  STRUCT
   S700_PLT : STRUCT 	//Temporary placeholder variable
    RACK0_PLT_CODE : INT ;
    RACK0_PLT_QTY : INT ;
    RACK0_PLT_PRIORITY : INT ;
    RACK0_HMI_PLT_CODE : INT ;
    RACK0_HMI_PLT_QTY : INT ;
    RACK1_PLT_CODE : INT ;
    RACK1_PLT_QTY : INT ;
    RACK1_PLT_PRIORITY : INT ;
    RACK1_HMI_PLT_CODE : INT ;
    RACK1_HMI_PLT_QTY : INT ;
    RACK2_PLT_CODE : INT ;
    RACK2_PLT_QTY : INT ;
    RACK2_PLT_PRIORITY : INT ;
    RACK2_HMI_PLT_CODE : INT ;
    RACK2_HMI_PLT_QTY : INT ;
    RACK3_PLT_CODE : INT ;
    RACK3_PLT_QTY : INT ;
    RACK3_PLT_PRIORITY : INT ;
    RACK3_HMI_PLT_CODE : INT ;
    RACK3_HMI_PLT_QTY : INT ;
    RACK4_PLT_CODE : INT ;
    RACK4_PLT_QTY : INT ;
    RACK4_PLT_PRIORITY : INT ;
    RACK4_HMI_PLT_CODE : INT ;
    RACK4_HMI_PLT_QTY : INT ;
    RACK5_PLT_CODE : INT ;
    RACK5_PLT_QTY : INT ;
    RACK5_PLT_PRIORITY : INT ;
    RACK5_HMI_PLT_CODE : INT ;
    RACK5_HMI_PLT_QTY : INT ;
    RACK6_PLT_CODE : INT ;
    RACK6_PLT_QTY : INT ;
    RACK6_PLT_PRIORITY : INT ;
    RACK6_HMI_PLT_CODE : INT ;
    RACK6_HMI_PLT_QTY : INT ;
    RACK7_PLT_CODE : INT ;
    RACK7_PLT_QTY : INT ;
    RACK7_PLT_PRIORITY : INT ;
    RACK7_HMI_PLT_CODE : INT ;
    RACK7_HMI_PLT_QTY : INT ;
    RACK8_PLT_CODE : INT ;
    RACK8_PLT_QTY : INT ;
    RACK8_PLT_PRIORITY : INT ;
    RACK8_HMI_PLT_CODE : INT ;
    RACK8_HMI_PLT_QTY : INT ;
    RACK9_PLT_CODE : INT ;
    RACK9_PLT_QTY : INT ;
    RACK9_PLT_PRIORITY : INT ;
    RACK9_HMI_PLT_CODE : INT ;
    RACK9_HMI_PLT_QTY : INT ;
    RACK10_PLT_CODE : INT ;
    RACK10_PLT_QTY : INT ;
    RACK10_PLT_PRIORITY : INT ;
    RACK10_HMI_PLT_CODE : INT ;
    RACK10_HMI_PLT_QTY : INT ;
    RACK11_PLT_CODE : INT ;
    RACK11_PLT_QTY : INT ;
    RACK11_PLT_PRIORITY : INT ;
    RACK11_HMI_PLT_CODE : INT ;
    RACK11_HMI_PLT_QTY : INT ;
    RACK12_PLT_CODE : INT ;
    RACK12_PLT_QTY : INT ;
    RACK12_PLT_PRIORITY : INT ;
    RACK12_HMI_PLT_CODE : INT ;
    RACK12_HMI_PLT_QTY : INT ;
   END_STRUCT ;
  END_STRUCT ;
BEGIN
   S700_PLT.RACK0_PLT_CODE := 0;
   S700_PLT.RACK0_PLT_QTY := 0;
   S700_PLT.RACK0_PLT_PRIORITY := 0;
   S700_PLT.RACK0_HMI_PLT_CODE := 0;
   S700_PLT.RACK0_HMI_PLT_QTY := 0;
   S700_PLT.RACK1_PLT_CODE := 0;
   S700_PLT.RACK1_PLT_QTY := 0;
   S700_PLT.RACK1_PLT_PRIORITY := 0;
   S700_PLT.RACK1_HMI_PLT_CODE := 0;
   S700_PLT.RACK1_HMI_PLT_QTY := 0;
   S700_PLT.RACK2_PLT_CODE := 0;
   S700_PLT.RACK2_PLT_QTY := 0;
   S700_PLT.RACK2_PLT_PRIORITY := 0;
   S700_PLT.RACK2_HMI_PLT_CODE := 0;
   S700_PLT.RACK2_HMI_PLT_QTY := 0;
   S700_PLT.RACK3_PLT_CODE := 0;
   S700_PLT.RACK3_PLT_QTY := 0;
   S700_PLT.RACK3_PLT_PRIORITY := 0;
   S700_PLT.RACK3_HMI_PLT_CODE := 0;
   S700_PLT.RACK3_HMI_PLT_QTY := 0;
   S700_PLT.RACK4_PLT_CODE := 0;
   S700_PLT.RACK4_PLT_QTY := 0;
   S700_PLT.RACK4_PLT_PRIORITY := 0;
   S700_PLT.RACK4_HMI_PLT_CODE := 0;
   S700_PLT.RACK4_HMI_PLT_QTY := 0;
   S700_PLT.RACK5_PLT_CODE := 0;
   S700_PLT.RACK5_PLT_QTY := 0;
   S700_PLT.RACK5_PLT_PRIORITY := 0;
   S700_PLT.RACK5_HMI_PLT_CODE := 0;
   S700_PLT.RACK5_HMI_PLT_QTY := 0;
   S700_PLT.RACK6_PLT_CODE := 0;
   S700_PLT.RACK6_PLT_QTY := 0;
   S700_PLT.RACK6_PLT_PRIORITY := 0;
   S700_PLT.RACK6_HMI_PLT_CODE := 0;
   S700_PLT.RACK6_HMI_PLT_QTY := 0;
   S700_PLT.RACK7_PLT_CODE := 0;
   S700_PLT.RACK7_PLT_QTY := 0;
   S700_PLT.RACK7_PLT_PRIORITY := 0;
   S700_PLT.RACK7_HMI_PLT_CODE := 0;
   S700_PLT.RACK7_HMI_PLT_QTY := 0;
   S700_PLT.RACK8_PLT_CODE := 0;
   S700_PLT.RACK8_PLT_QTY := 0;
   S700_PLT.RACK8_PLT_PRIORITY := 0;
   S700_PLT.RACK8_HMI_PLT_CODE := 0;
   S700_PLT.RACK8_HMI_PLT_QTY := 0;
   S700_PLT.RACK9_PLT_CODE := 0;
   S700_PLT.RACK9_PLT_QTY := 0;
   S700_PLT.RACK9_PLT_PRIORITY := 0;
   S700_PLT.RACK9_HMI_PLT_CODE := 0;
   S700_PLT.RACK9_HMI_PLT_QTY := 0;
   S700_PLT.RACK10_PLT_CODE := 0;
   S700_PLT.RACK10_PLT_QTY := 0;
   S700_PLT.RACK10_PLT_PRIORITY := 0;
   S700_PLT.RACK10_HMI_PLT_CODE := 0;
   S700_PLT.RACK10_HMI_PLT_QTY := 0;
   S700_PLT.RACK11_PLT_CODE := 0;
   S700_PLT.RACK11_PLT_QTY := 0;
   S700_PLT.RACK11_PLT_PRIORITY := 0;
   S700_PLT.RACK11_HMI_PLT_CODE := 0;
   S700_PLT.RACK11_HMI_PLT_QTY := 0;
   S700_PLT.RACK12_PLT_CODE := 0;
   S700_PLT.RACK12_PLT_QTY := 0;
   S700_PLT.RACK12_PLT_PRIORITY := 0;
   S700_PLT.RACK12_HMI_PLT_CODE := 0;
   S700_PLT.RACK12_HMI_PLT_QTY := 0;
END_DATA_BLOCK

DATA_BLOCK DB 60
TITLE =
VERSION : 0.1


  STRUCT
   FC1_SEND_1 : ARRAY  [0 .. 699 ] OF BYTE  := B#16#0;
  END_STRUCT ;
BEGIN
   FC1_SEND_1[0] := B#16#0;
   FC1_SEND_1[1] := B#16#0;
   FC1_SEND_1[2] := B#16#0;
   FC1_SEND_1[3] := B#16#0;
   FC1_SEND_1[4] := B#16#0;
   FC1_SEND_1[5] := B#16#0;
   FC1_SEND_1[6] := B#16#0;
   FC1_SEND_1[7] := B#16#0;
   FC1_SEND_1[8] := B#16#0;
   FC1_SEND_1[9] := B#16#0;
   FC1_SEND_1[10] := B#16#0;
   FC1_SEND_1[11] := B#16#0;
   FC1_SEND_1[12] := B#16#0;
   FC1_SEND_1[13] := B#16#0;
   FC1_SEND_1[14] := B#16#0;
   FC1_SEND_1[15] := B#16#0;
   FC1_SEND_1[16] := B#16#0;
   FC1_SEND_1[17] := B#16#0;
   FC1_SEND_1[18] := B#16#0;
   FC1_SEND_1[19] := B#16#0;
   FC1_SEND_1[20] := B#16#0;
   FC1_SEND_1[21] := B#16#0;
   FC1_SEND_1[22] := B#16#0;
   FC1_SEND_1[23] := B#16#0;
   FC1_SEND_1[24] := B#16#0;
   FC1_SEND_1[25] := B#16#0;
   FC1_SEND_1[26] := B#16#0;
   FC1_SEND_1[27] := B#16#0;
   FC1_SEND_1[28] := B#16#0;
   FC1_SEND_1[29] := B#16#0;
   FC1_SEND_1[30] := B#16#0;
   FC1_SEND_1[31] := B#16#0;
   FC1_SEND_1[32] := B#16#0;
   FC1_SEND_1[33] := B#16#0;
   FC1_SEND_1[34] := B#16#0;
   FC1_SEND_1[35] := B#16#0;
   FC1_SEND_1[36] := B#16#0;
   FC1_SEND_1[37] := B#16#0;
   FC1_SEND_1[38] := B#16#0;
   FC1_SEND_1[39] := B#16#0;
   FC1_SEND_1[40] := B#16#0;
   FC1_SEND_1[41] := B#16#0;
   FC1_SEND_1[42] := B#16#0;
   FC1_SEND_1[43] := B#16#0;
   FC1_SEND_1[44] := B#16#0;
   FC1_SEND_1[45] := B#16#0;
   FC1_SEND_1[46] := B#16#0;
   FC1_SEND_1[47] := B#16#0;
   FC1_SEND_1[48] := B#16#0;
   FC1_SEND_1[49] := B#16#0;
   FC1_SEND_1[50] := B#16#0;
   FC1_SEND_1[51] := B#16#0;
   FC1_SEND_1[52] := B#16#0;
   FC1_SEND_1[53] := B#16#0;
   FC1_SEND_1[54] := B#16#0;
   FC1_SEND_1[55] := B#16#0;
   FC1_SEND_1[56] := B#16#0;
   FC1_SEND_1[57] := B#16#0;
   FC1_SEND_1[58] := B#16#0;
   FC1_SEND_1[59] := B#16#0;
   FC1_SEND_1[60] := B#16#0;
   FC1_SEND_1[61] := B#16#0;
   FC1_SEND_1[62] := B#16#0;
   FC1_SEND_1[63] := B#16#0;
   FC1_SEND_1[64] := B#16#0;
   FC1_SEND_1[65] := B#16#0;
   FC1_SEND_1[66] := B#16#0;
   FC1_SEND_1[67] := B#16#0;
   FC1_SEND_1[68] := B#16#0;
   FC1_SEND_1[69] := B#16#0;
   FC1_SEND_1[70] := B#16#0;
   FC1_SEND_1[71] := B#16#0;
   FC1_SEND_1[72] := B#16#0;
   FC1_SEND_1[73] := B#16#0;
   FC1_SEND_1[74] := B#16#0;
   FC1_SEND_1[75] := B#16#0;
   FC1_SEND_1[76] := B#16#0;
   FC1_SEND_1[77] := B#16#0;
   FC1_SEND_1[78] := B#16#0;
   FC1_SEND_1[79] := B#16#0;
   FC1_SEND_1[80] := B#16#0;
   FC1_SEND_1[81] := B#16#0;
   FC1_SEND_1[82] := B#16#0;
   FC1_SEND_1[83] := B#16#0;
   FC1_SEND_1[84] := B#16#0;
   FC1_SEND_1[85] := B#16#0;
   FC1_SEND_1[86] := B#16#0;
   FC1_SEND_1[87] := B#16#0;
   FC1_SEND_1[88] := B#16#0;
   FC1_SEND_1[89] := B#16#0;
   FC1_SEND_1[90] := B#16#0;
   FC1_SEND_1[91] := B#16#0;
   FC1_SEND_1[92] := B#16#0;
   FC1_SEND_1[93] := B#16#0;
   FC1_SEND_1[94] := B#16#0;
   FC1_SEND_1[95] := B#16#0;
   FC1_SEND_1[96] := B#16#0;
   FC1_SEND_1[97] := B#16#0;
   FC1_SEND_1[98] := B#16#0;
   FC1_SEND_1[99] := B#16#0;
   FC1_SEND_1[100] := B#16#0;
   FC1_SEND_1[101] := B#16#0;
   FC1_SEND_1[102] := B#16#0;
   FC1_SEND_1[103] := B#16#0;
   FC1_SEND_1[104] := B#16#0;
   FC1_SEND_1[105] := B#16#0;
   FC1_SEND_1[106] := B#16#0;
   FC1_SEND_1[107] := B#16#0;
   FC1_SEND_1[108] := B#16#0;
   FC1_SEND_1[109] := B#16#0;
   FC1_SEND_1[110] := B#16#0;
   FC1_SEND_1[111] := B#16#0;
   FC1_SEND_1[112] := B#16#0;
   FC1_SEND_1[113] := B#16#0;
   FC1_SEND_1[114] := B#16#0;
   FC1_SEND_1[115] := B#16#0;
   FC1_SEND_1[116] := B#16#0;
   FC1_SEND_1[117] := B#16#0;
   FC1_SEND_1[118] := B#16#0;
   FC1_SEND_1[119] := B#16#0;
   FC1_SEND_1[120] := B#16#0;
   FC1_SEND_1[121] := B#16#0;
   FC1_SEND_1[122] := B#16#0;
   FC1_SEND_1[123] := B#16#0;
   FC1_SEND_1[124] := B#16#0;
   FC1_SEND_1[125] := B#16#0;
   FC1_SEND_1[126] := B#16#0;
   FC1_SEND_1[127] := B#16#0;
   FC1_SEND_1[128] := B#16#0;
   FC1_SEND_1[129] := B#16#0;
   FC1_SEND_1[130] := B#16#0;
   FC1_SEND_1[131] := B#16#0;
   FC1_SEND_1[132] := B#16#0;
   FC1_SEND_1[133] := B#16#0;
   FC1_SEND_1[134] := B#16#0;
   FC1_SEND_1[135] := B#16#0;
   FC1_SEND_1[136] := B#16#0;
   FC1_SEND_1[137] := B#16#0;
   FC1_SEND_1[138] := B#16#0;
   FC1_SEND_1[139] := B#16#0;
   FC1_SEND_1[140] := B#16#0;
   FC1_SEND_1[141] := B#16#0;
   FC1_SEND_1[142] := B#16#0;
   FC1_SEND_1[143] := B#16#0;
   FC1_SEND_1[144] := B#16#0;
   FC1_SEND_1[145] := B#16#0;
   FC1_SEND_1[146] := B#16#0;
   FC1_SEND_1[147] := B#16#0;
   FC1_SEND_1[148] := B#16#0;
   FC1_SEND_1[149] := B#16#0;
   FC1_SEND_1[150] := B#16#0;
   FC1_SEND_1[151] := B#16#0;
   FC1_SEND_1[152] := B#16#0;
   FC1_SEND_1[153] := B#16#0;
   FC1_SEND_1[154] := B#16#0;
   FC1_SEND_1[155] := B#16#0;
   FC1_SEND_1[156] := B#16#0;
   FC1_SEND_1[157] := B#16#0;
   FC1_SEND_1[158] := B#16#0;
   FC1_SEND_1[159] := B#16#0;
   FC1_SEND_1[160] := B#16#0;
   FC1_SEND_1[161] := B#16#0;
   FC1_SEND_1[162] := B#16#0;
   FC1_SEND_1[163] := B#16#0;
   FC1_SEND_1[164] := B#16#0;
   FC1_SEND_1[165] := B#16#0;
   FC1_SEND_1[166] := B#16#0;
   FC1_SEND_1[167] := B#16#0;
   FC1_SEND_1[168] := B#16#0;
   FC1_SEND_1[169] := B#16#0;
   FC1_SEND_1[170] := B#16#0;
   FC1_SEND_1[171] := B#16#0;
   FC1_SEND_1[172] := B#16#0;
   FC1_SEND_1[173] := B#16#0;
   FC1_SEND_1[174] := B#16#0;
   FC1_SEND_1[175] := B#16#0;
   FC1_SEND_1[176] := B#16#0;
   FC1_SEND_1[177] := B#16#0;
   FC1_SEND_1[178] := B#16#0;
   FC1_SEND_1[179] := B#16#0;
   FC1_SEND_1[180] := B#16#0;
   FC1_SEND_1[181] := B#16#0;
   FC1_SEND_1[182] := B#16#0;
   FC1_SEND_1[183] := B#16#0;
   FC1_SEND_1[184] := B#16#0;
   FC1_SEND_1[185] := B#16#0;
   FC1_SEND_1[186] := B#16#0;
   FC1_SEND_1[187] := B#16#0;
   FC1_SEND_1[188] := B#16#0;
   FC1_SEND_1[189] := B#16#0;
   FC1_SEND_1[190] := B#16#0;
   FC1_SEND_1[191] := B#16#0;
   FC1_SEND_1[192] := B#16#0;
   FC1_SEND_1[193] := B#16#0;
   FC1_SEND_1[194] := B#16#0;
   FC1_SEND_1[195] := B#16#0;
   FC1_SEND_1[196] := B#16#0;
   FC1_SEND_1[197] := B#16#0;
   FC1_SEND_1[198] := B#16#0;
   FC1_SEND_1[199] := B#16#0;
   FC1_SEND_1[200] := B#16#0;
   FC1_SEND_1[201] := B#16#0;
   FC1_SEND_1[202] := B#16#0;
   FC1_SEND_1[203] := B#16#0;
   FC1_SEND_1[204] := B#16#0;
   FC1_SEND_1[205] := B#16#0;
   FC1_SEND_1[206] := B#16#0;
   FC1_SEND_1[207] := B#16#0;
   FC1_SEND_1[208] := B#16#0;
   FC1_SEND_1[209] := B#16#0;
   FC1_SEND_1[210] := B#16#0;
   FC1_SEND_1[211] := B#16#0;
   FC1_SEND_1[212] := B#16#0;
   FC1_SEND_1[213] := B#16#0;
   FC1_SEND_1[214] := B#16#0;
   FC1_SEND_1[215] := B#16#0;
   FC1_SEND_1[216] := B#16#0;
   FC1_SEND_1[217] := B#16#0;
   FC1_SEND_1[218] := B#16#0;
   FC1_SEND_1[219] := B#16#0;
   FC1_SEND_1[220] := B#16#0;
   FC1_SEND_1[221] := B#16#0;
   FC1_SEND_1[222] := B#16#0;
   FC1_SEND_1[223] := B#16#0;
   FC1_SEND_1[224] := B#16#0;
   FC1_SEND_1[225] := B#16#0;
   FC1_SEND_1[226] := B#16#0;
   FC1_SEND_1[227] := B#16#0;
   FC1_SEND_1[228] := B#16#0;
   FC1_SEND_1[229] := B#16#0;
   FC1_SEND_1[230] := B#16#0;
   FC1_SEND_1[231] := B#16#0;
   FC1_SEND_1[232] := B#16#0;
   FC1_SEND_1[233] := B#16#0;
   FC1_SEND_1[234] := B#16#0;
   FC1_SEND_1[235] := B#16#0;
   FC1_SEND_1[236] := B#16#0;
   FC1_SEND_1[237] := B#16#0;
   FC1_SEND_1[238] := B#16#0;
   FC1_SEND_1[239] := B#16#0;
   FC1_SEND_1[240] := B#16#0;
   FC1_SEND_1[241] := B#16#0;
   FC1_SEND_1[242] := B#16#0;
   FC1_SEND_1[243] := B#16#0;
   FC1_SEND_1[244] := B#16#0;
   FC1_SEND_1[245] := B#16#0;
   FC1_SEND_1[246] := B#16#0;
   FC1_SEND_1[247] := B#16#0;
   FC1_SEND_1[248] := B#16#0;
   FC1_SEND_1[249] := B#16#0;
   FC1_SEND_1[250] := B#16#0;
   FC1_SEND_1[251] := B#16#0;
   FC1_SEND_1[252] := B#16#0;
   FC1_SEND_1[253] := B#16#0;
   FC1_SEND_1[254] := B#16#0;
   FC1_SEND_1[255] := B#16#0;
   FC1_SEND_1[256] := B#16#0;
   FC1_SEND_1[257] := B#16#0;
   FC1_SEND_1[258] := B#16#0;
   FC1_SEND_1[259] := B#16#0;
   FC1_SEND_1[260] := B#16#0;
   FC1_SEND_1[261] := B#16#0;
   FC1_SEND_1[262] := B#16#0;
   FC1_SEND_1[263] := B#16#0;
   FC1_SEND_1[264] := B#16#0;
   FC1_SEND_1[265] := B#16#0;
   FC1_SEND_1[266] := B#16#0;
   FC1_SEND_1[267] := B#16#0;
   FC1_SEND_1[268] := B#16#0;
   FC1_SEND_1[269] := B#16#0;
   FC1_SEND_1[270] := B#16#0;
   FC1_SEND_1[271] := B#16#0;
   FC1_SEND_1[272] := B#16#0;
   FC1_SEND_1[273] := B#16#0;
   FC1_SEND_1[274] := B#16#0;
   FC1_SEND_1[275] := B#16#0;
   FC1_SEND_1[276] := B#16#0;
   FC1_SEND_1[277] := B#16#0;
   FC1_SEND_1[278] := B#16#0;
   FC1_SEND_1[279] := B#16#0;
   FC1_SEND_1[280] := B#16#0;
   FC1_SEND_1[281] := B#16#0;
   FC1_SEND_1[282] := B#16#0;
   FC1_SEND_1[283] := B#16#0;
   FC1_SEND_1[284] := B#16#0;
   FC1_SEND_1[285] := B#16#0;
   FC1_SEND_1[286] := B#16#0;
   FC1_SEND_1[287] := B#16#0;
   FC1_SEND_1[288] := B#16#0;
   FC1_SEND_1[289] := B#16#0;
   FC1_SEND_1[290] := B#16#0;
   FC1_SEND_1[291] := B#16#0;
   FC1_SEND_1[292] := B#16#0;
   FC1_SEND_1[293] := B#16#0;
   FC1_SEND_1[294] := B#16#0;
   FC1_SEND_1[295] := B#16#0;
   FC1_SEND_1[296] := B#16#0;
   FC1_SEND_1[297] := B#16#0;
   FC1_SEND_1[298] := B#16#0;
   FC1_SEND_1[299] := B#16#0;
   FC1_SEND_1[300] := B#16#0;
   FC1_SEND_1[301] := B#16#0;
   FC1_SEND_1[302] := B#16#0;
   FC1_SEND_1[303] := B#16#0;
   FC1_SEND_1[304] := B#16#0;
   FC1_SEND_1[305] := B#16#0;
   FC1_SEND_1[306] := B#16#0;
   FC1_SEND_1[307] := B#16#0;
   FC1_SEND_1[308] := B#16#0;
   FC1_SEND_1[309] := B#16#0;
   FC1_SEND_1[310] := B#16#0;
   FC1_SEND_1[311] := B#16#0;
   FC1_SEND_1[312] := B#16#0;
   FC1_SEND_1[313] := B#16#0;
   FC1_SEND_1[314] := B#16#0;
   FC1_SEND_1[315] := B#16#0;
   FC1_SEND_1[316] := B#16#0;
   FC1_SEND_1[317] := B#16#0;
   FC1_SEND_1[318] := B#16#0;
   FC1_SEND_1[319] := B#16#0;
   FC1_SEND_1[320] := B#16#0;
   FC1_SEND_1[321] := B#16#0;
   FC1_SEND_1[322] := B#16#0;
   FC1_SEND_1[323] := B#16#0;
   FC1_SEND_1[324] := B#16#0;
   FC1_SEND_1[325] := B#16#0;
   FC1_SEND_1[326] := B#16#0;
   FC1_SEND_1[327] := B#16#0;
   FC1_SEND_1[328] := B#16#0;
   FC1_SEND_1[329] := B#16#0;
   FC1_SEND_1[330] := B#16#0;
   FC1_SEND_1[331] := B#16#0;
   FC1_SEND_1[332] := B#16#0;
   FC1_SEND_1[333] := B#16#0;
   FC1_SEND_1[334] := B#16#0;
   FC1_SEND_1[335] := B#16#0;
   FC1_SEND_1[336] := B#16#0;
   FC1_SEND_1[337] := B#16#0;
   FC1_SEND_1[338] := B#16#0;
   FC1_SEND_1[339] := B#16#0;
   FC1_SEND_1[340] := B#16#0;
   FC1_SEND_1[341] := B#16#0;
   FC1_SEND_1[342] := B#16#0;
   FC1_SEND_1[343] := B#16#0;
   FC1_SEND_1[344] := B#16#0;
   FC1_SEND_1[345] := B#16#0;
   FC1_SEND_1[346] := B#16#0;
   FC1_SEND_1[347] := B#16#0;
   FC1_SEND_1[348] := B#16#0;
   FC1_SEND_1[349] := B#16#0;
   FC1_SEND_1[350] := B#16#0;
   FC1_SEND_1[351] := B#16#0;
   FC1_SEND_1[352] := B#16#0;
   FC1_SEND_1[353] := B#16#0;
   FC1_SEND_1[354] := B#16#0;
   FC1_SEND_1[355] := B#16#0;
   FC1_SEND_1[356] := B#16#0;
   FC1_SEND_1[357] := B#16#0;
   FC1_SEND_1[358] := B#16#0;
   FC1_SEND_1[359] := B#16#0;
   FC1_SEND_1[360] := B#16#0;
   FC1_SEND_1[361] := B#16#0;
   FC1_SEND_1[362] := B#16#0;
   FC1_SEND_1[363] := B#16#0;
   FC1_SEND_1[364] := B#16#0;
   FC1_SEND_1[365] := B#16#0;
   FC1_SEND_1[366] := B#16#0;
   FC1_SEND_1[367] := B#16#0;
   FC1_SEND_1[368] := B#16#0;
   FC1_SEND_1[369] := B#16#0;
   FC1_SEND_1[370] := B#16#0;
   FC1_SEND_1[371] := B#16#0;
   FC1_SEND_1[372] := B#16#0;
   FC1_SEND_1[373] := B#16#0;
   FC1_SEND_1[374] := B#16#0;
   FC1_SEND_1[375] := B#16#0;
   FC1_SEND_1[376] := B#16#0;
   FC1_SEND_1[377] := B#16#0;
   FC1_SEND_1[378] := B#16#0;
   FC1_SEND_1[379] := B#16#0;
   FC1_SEND_1[380] := B#16#0;
   FC1_SEND_1[381] := B#16#0;
   FC1_SEND_1[382] := B#16#0;
   FC1_SEND_1[383] := B#16#0;
   FC1_SEND_1[384] := B#16#0;
   FC1_SEND_1[385] := B#16#0;
   FC1_SEND_1[386] := B#16#0;
   FC1_SEND_1[387] := B#16#0;
   FC1_SEND_1[388] := B#16#0;
   FC1_SEND_1[389] := B#16#0;
   FC1_SEND_1[390] := B#16#0;
   FC1_SEND_1[391] := B#16#0;
   FC1_SEND_1[392] := B#16#0;
   FC1_SEND_1[393] := B#16#0;
   FC1_SEND_1[394] := B#16#0;
   FC1_SEND_1[395] := B#16#0;
   FC1_SEND_1[396] := B#16#0;
   FC1_SEND_1[397] := B#16#0;
   FC1_SEND_1[398] := B#16#0;
   FC1_SEND_1[399] := B#16#0;
   FC1_SEND_1[400] := B#16#0;
   FC1_SEND_1[401] := B#16#0;
   FC1_SEND_1[402] := B#16#0;
   FC1_SEND_1[403] := B#16#0;
   FC1_SEND_1[404] := B#16#0;
   FC1_SEND_1[405] := B#16#0;
   FC1_SEND_1[406] := B#16#0;
   FC1_SEND_1[407] := B#16#0;
   FC1_SEND_1[408] := B#16#0;
   FC1_SEND_1[409] := B#16#0;
   FC1_SEND_1[410] := B#16#0;
   FC1_SEND_1[411] := B#16#0;
   FC1_SEND_1[412] := B#16#0;
   FC1_SEND_1[413] := B#16#0;
   FC1_SEND_1[414] := B#16#0;
   FC1_SEND_1[415] := B#16#0;
   FC1_SEND_1[416] := B#16#0;
   FC1_SEND_1[417] := B#16#0;
   FC1_SEND_1[418] := B#16#0;
   FC1_SEND_1[419] := B#16#0;
   FC1_SEND_1[420] := B#16#0;
   FC1_SEND_1[421] := B#16#0;
   FC1_SEND_1[422] := B#16#0;
   FC1_SEND_1[423] := B#16#0;
   FC1_SEND_1[424] := B#16#0;
   FC1_SEND_1[425] := B#16#0;
   FC1_SEND_1[426] := B#16#0;
   FC1_SEND_1[427] := B#16#0;
   FC1_SEND_1[428] := B#16#0;
   FC1_SEND_1[429] := B#16#0;
   FC1_SEND_1[430] := B#16#0;
   FC1_SEND_1[431] := B#16#0;
   FC1_SEND_1[432] := B#16#0;
   FC1_SEND_1[433] := B#16#0;
   FC1_SEND_1[434] := B#16#0;
   FC1_SEND_1[435] := B#16#0;
   FC1_SEND_1[436] := B#16#0;
   FC1_SEND_1[437] := B#16#0;
   FC1_SEND_1[438] := B#16#0;
   FC1_SEND_1[439] := B#16#0;
   FC1_SEND_1[440] := B#16#0;
   FC1_SEND_1[441] := B#16#0;
   FC1_SEND_1[442] := B#16#0;
   FC1_SEND_1[443] := B#16#0;
   FC1_SEND_1[444] := B#16#0;
   FC1_SEND_1[445] := B#16#0;
   FC1_SEND_1[446] := B#16#0;
   FC1_SEND_1[447] := B#16#0;
   FC1_SEND_1[448] := B#16#0;
   FC1_SEND_1[449] := B#16#0;
   FC1_SEND_1[450] := B#16#0;
   FC1_SEND_1[451] := B#16#0;
   FC1_SEND_1[452] := B#16#0;
   FC1_SEND_1[453] := B#16#0;
   FC1_SEND_1[454] := B#16#0;
   FC1_SEND_1[455] := B#16#0;
   FC1_SEND_1[456] := B#16#0;
   FC1_SEND_1[457] := B#16#0;
   FC1_SEND_1[458] := B#16#0;
   FC1_SEND_1[459] := B#16#0;
   FC1_SEND_1[460] := B#16#0;
   FC1_SEND_1[461] := B#16#0;
   FC1_SEND_1[462] := B#16#0;
   FC1_SEND_1[463] := B#16#0;
   FC1_SEND_1[464] := B#16#0;
   FC1_SEND_1[465] := B#16#0;
   FC1_SEND_1[466] := B#16#0;
   FC1_SEND_1[467] := B#16#0;
   FC1_SEND_1[468] := B#16#0;
   FC1_SEND_1[469] := B#16#0;
   FC1_SEND_1[470] := B#16#0;
   FC1_SEND_1[471] := B#16#0;
   FC1_SEND_1[472] := B#16#0;
   FC1_SEND_1[473] := B#16#0;
   FC1_SEND_1[474] := B#16#0;
   FC1_SEND_1[475] := B#16#0;
   FC1_SEND_1[476] := B#16#0;
   FC1_SEND_1[477] := B#16#0;
   FC1_SEND_1[478] := B#16#0;
   FC1_SEND_1[479] := B#16#0;
   FC1_SEND_1[480] := B#16#0;
   FC1_SEND_1[481] := B#16#0;
   FC1_SEND_1[482] := B#16#0;
   FC1_SEND_1[483] := B#16#0;
   FC1_SEND_1[484] := B#16#0;
   FC1_SEND_1[485] := B#16#0;
   FC1_SEND_1[486] := B#16#0;
   FC1_SEND_1[487] := B#16#0;
   FC1_SEND_1[488] := B#16#0;
   FC1_SEND_1[489] := B#16#0;
   FC1_SEND_1[490] := B#16#0;
   FC1_SEND_1[491] := B#16#0;
   FC1_SEND_1[492] := B#16#0;
   FC1_SEND_1[493] := B#16#0;
   FC1_SEND_1[494] := B#16#0;
   FC1_SEND_1[495] := B#16#0;
   FC1_SEND_1[496] := B#16#0;
   FC1_SEND_1[497] := B#16#0;
   FC1_SEND_1[498] := B#16#0;
   FC1_SEND_1[499] := B#16#0;
   FC1_SEND_1[500] := B#16#0;
   FC1_SEND_1[501] := B#16#0;
   FC1_SEND_1[502] := B#16#0;
   FC1_SEND_1[503] := B#16#0;
   FC1_SEND_1[504] := B#16#0;
   FC1_SEND_1[505] := B#16#0;
   FC1_SEND_1[506] := B#16#0;
   FC1_SEND_1[507] := B#16#0;
   FC1_SEND_1[508] := B#16#0;
   FC1_SEND_1[509] := B#16#0;
   FC1_SEND_1[510] := B#16#0;
   FC1_SEND_1[511] := B#16#0;
   FC1_SEND_1[512] := B#16#0;
   FC1_SEND_1[513] := B#16#0;
   FC1_SEND_1[514] := B#16#0;
   FC1_SEND_1[515] := B#16#0;
   FC1_SEND_1[516] := B#16#0;
   FC1_SEND_1[517] := B#16#0;
   FC1_SEND_1[518] := B#16#0;
   FC1_SEND_1[519] := B#16#0;
   FC1_SEND_1[520] := B#16#0;
   FC1_SEND_1[521] := B#16#0;
   FC1_SEND_1[522] := B#16#0;
   FC1_SEND_1[523] := B#16#0;
   FC1_SEND_1[524] := B#16#0;
   FC1_SEND_1[525] := B#16#0;
   FC1_SEND_1[526] := B#16#0;
   FC1_SEND_1[527] := B#16#0;
   FC1_SEND_1[528] := B#16#0;
   FC1_SEND_1[529] := B#16#0;
   FC1_SEND_1[530] := B#16#0;
   FC1_SEND_1[531] := B#16#0;
   FC1_SEND_1[532] := B#16#0;
   FC1_SEND_1[533] := B#16#0;
   FC1_SEND_1[534] := B#16#0;
   FC1_SEND_1[535] := B#16#0;
   FC1_SEND_1[536] := B#16#0;
   FC1_SEND_1[537] := B#16#0;
   FC1_SEND_1[538] := B#16#0;
   FC1_SEND_1[539] := B#16#0;
   FC1_SEND_1[540] := B#16#0;
   FC1_SEND_1[541] := B#16#0;
   FC1_SEND_1[542] := B#16#0;
   FC1_SEND_1[543] := B#16#0;
   FC1_SEND_1[544] := B#16#0;
   FC1_SEND_1[545] := B#16#0;
   FC1_SEND_1[546] := B#16#0;
   FC1_SEND_1[547] := B#16#0;
   FC1_SEND_1[548] := B#16#0;
   FC1_SEND_1[549] := B#16#0;
   FC1_SEND_1[550] := B#16#0;
   FC1_SEND_1[551] := B#16#0;
   FC1_SEND_1[552] := B#16#0;
   FC1_SEND_1[553] := B#16#0;
   FC1_SEND_1[554] := B#16#0;
   FC1_SEND_1[555] := B#16#0;
   FC1_SEND_1[556] := B#16#0;
   FC1_SEND_1[557] := B#16#0;
   FC1_SEND_1[558] := B#16#0;
   FC1_SEND_1[559] := B#16#0;
   FC1_SEND_1[560] := B#16#0;
   FC1_SEND_1[561] := B#16#0;
   FC1_SEND_1[562] := B#16#0;
   FC1_SEND_1[563] := B#16#0;
   FC1_SEND_1[564] := B#16#0;
   FC1_SEND_1[565] := B#16#0;
   FC1_SEND_1[566] := B#16#0;
   FC1_SEND_1[567] := B#16#0;
   FC1_SEND_1[568] := B#16#0;
   FC1_SEND_1[569] := B#16#0;
   FC1_SEND_1[570] := B#16#0;
   FC1_SEND_1[571] := B#16#0;
   FC1_SEND_1[572] := B#16#0;
   FC1_SEND_1[573] := B#16#0;
   FC1_SEND_1[574] := B#16#0;
   FC1_SEND_1[575] := B#16#0;
   FC1_SEND_1[576] := B#16#0;
   FC1_SEND_1[577] := B#16#0;
   FC1_SEND_1[578] := B#16#0;
   FC1_SEND_1[579] := B#16#0;
   FC1_SEND_1[580] := B#16#0;
   FC1_SEND_1[581] := B#16#0;
   FC1_SEND_1[582] := B#16#0;
   FC1_SEND_1[583] := B#16#0;
   FC1_SEND_1[584] := B#16#0;
   FC1_SEND_1[585] := B#16#0;
   FC1_SEND_1[586] := B#16#0;
   FC1_SEND_1[587] := B#16#0;
   FC1_SEND_1[588] := B#16#0;
   FC1_SEND_1[589] := B#16#0;
   FC1_SEND_1[590] := B#16#0;
   FC1_SEND_1[591] := B#16#0;
   FC1_SEND_1[592] := B#16#0;
   FC1_SEND_1[593] := B#16#0;
   FC1_SEND_1[594] := B#16#0;
   FC1_SEND_1[595] := B#16#0;
   FC1_SEND_1[596] := B#16#0;
   FC1_SEND_1[597] := B#16#0;
   FC1_SEND_1[598] := B#16#0;
   FC1_SEND_1[599] := B#16#0;
   FC1_SEND_1[600] := B#16#0;
   FC1_SEND_1[601] := B#16#0;
   FC1_SEND_1[602] := B#16#0;
   FC1_SEND_1[603] := B#16#0;
   FC1_SEND_1[604] := B#16#0;
   FC1_SEND_1[605] := B#16#0;
   FC1_SEND_1[606] := B#16#0;
   FC1_SEND_1[607] := B#16#0;
   FC1_SEND_1[608] := B#16#0;
   FC1_SEND_1[609] := B#16#0;
   FC1_SEND_1[610] := B#16#0;
   FC1_SEND_1[611] := B#16#0;
   FC1_SEND_1[612] := B#16#0;
   FC1_SEND_1[613] := B#16#0;
   FC1_SEND_1[614] := B#16#0;
   FC1_SEND_1[615] := B#16#0;
   FC1_SEND_1[616] := B#16#0;
   FC1_SEND_1[617] := B#16#0;
   FC1_SEND_1[618] := B#16#0;
   FC1_SEND_1[619] := B#16#0;
   FC1_SEND_1[620] := B#16#0;
   FC1_SEND_1[621] := B#16#0;
   FC1_SEND_1[622] := B#16#0;
   FC1_SEND_1[623] := B#16#0;
   FC1_SEND_1[624] := B#16#0;
   FC1_SEND_1[625] := B#16#0;
   FC1_SEND_1[626] := B#16#0;
   FC1_SEND_1[627] := B#16#0;
   FC1_SEND_1[628] := B#16#0;
   FC1_SEND_1[629] := B#16#0;
   FC1_SEND_1[630] := B#16#0;
   FC1_SEND_1[631] := B#16#0;
   FC1_SEND_1[632] := B#16#0;
   FC1_SEND_1[633] := B#16#0;
   FC1_SEND_1[634] := B#16#0;
   FC1_SEND_1[635] := B#16#0;
   FC1_SEND_1[636] := B#16#0;
   FC1_SEND_1[637] := B#16#0;
   FC1_SEND_1[638] := B#16#0;
   FC1_SEND_1[639] := B#16#0;
   FC1_SEND_1[640] := B#16#0;
   FC1_SEND_1[641] := B#16#0;
   FC1_SEND_1[642] := B#16#0;
   FC1_SEND_1[643] := B#16#0;
   FC1_SEND_1[644] := B#16#0;
   FC1_SEND_1[645] := B#16#0;
   FC1_SEND_1[646] := B#16#0;
   FC1_SEND_1[647] := B#16#0;
   FC1_SEND_1[648] := B#16#0;
   FC1_SEND_1[649] := B#16#0;
   FC1_SEND_1[650] := B#16#0;
   FC1_SEND_1[651] := B#16#0;
   FC1_SEND_1[652] := B#16#0;
   FC1_SEND_1[653] := B#16#0;
   FC1_SEND_1[654] := B#16#0;
   FC1_SEND_1[655] := B#16#0;
   FC1_SEND_1[656] := B#16#0;
   FC1_SEND_1[657] := B#16#0;
   FC1_SEND_1[658] := B#16#0;
   FC1_SEND_1[659] := B#16#0;
   FC1_SEND_1[660] := B#16#0;
   FC1_SEND_1[661] := B#16#0;
   FC1_SEND_1[662] := B#16#0;
   FC1_SEND_1[663] := B#16#0;
   FC1_SEND_1[664] := B#16#0;
   FC1_SEND_1[665] := B#16#0;
   FC1_SEND_1[666] := B#16#0;
   FC1_SEND_1[667] := B#16#0;
   FC1_SEND_1[668] := B#16#0;
   FC1_SEND_1[669] := B#16#0;
   FC1_SEND_1[670] := B#16#0;
   FC1_SEND_1[671] := B#16#0;
   FC1_SEND_1[672] := B#16#0;
   FC1_SEND_1[673] := B#16#0;
   FC1_SEND_1[674] := B#16#0;
   FC1_SEND_1[675] := B#16#0;
   FC1_SEND_1[676] := B#16#0;
   FC1_SEND_1[677] := B#16#0;
   FC1_SEND_1[678] := B#16#0;
   FC1_SEND_1[679] := B#16#0;
   FC1_SEND_1[680] := B#16#0;
   FC1_SEND_1[681] := B#16#0;
   FC1_SEND_1[682] := B#16#0;
   FC1_SEND_1[683] := B#16#0;
   FC1_SEND_1[684] := B#16#0;
   FC1_SEND_1[685] := B#16#0;
   FC1_SEND_1[686] := B#16#0;
   FC1_SEND_1[687] := B#16#0;
   FC1_SEND_1[688] := B#16#0;
   FC1_SEND_1[689] := B#16#0;
   FC1_SEND_1[690] := B#16#0;
   FC1_SEND_1[691] := B#16#0;
   FC1_SEND_1[692] := B#16#0;
   FC1_SEND_1[693] := B#16#0;
   FC1_SEND_1[694] := B#16#0;
   FC1_SEND_1[695] := B#16#0;
   FC1_SEND_1[696] := B#16#0;
   FC1_SEND_1[697] := B#16#0;
   FC1_SEND_1[698] := B#16#0;
   FC1_SEND_1[699] := B#16#0;
END_DATA_BLOCK

DATA_BLOCK DB 61
TITLE =
VERSION : 0.1


  STRUCT
   FC2_RECV_1 : ARRAY  [0 .. 699 ] OF BYTE  := B#16#0;
  END_STRUCT ;
BEGIN
   FC2_RECV_1[0] := B#16#0;
   FC2_RECV_1[1] := B#16#0;
   FC2_RECV_1[2] := B#16#0;
   FC2_RECV_1[3] := B#16#0;
   FC2_RECV_1[4] := B#16#0;
   FC2_RECV_1[5] := B#16#0;
   FC2_RECV_1[6] := B#16#0;
   FC2_RECV_1[7] := B#16#0;
   FC2_RECV_1[8] := B#16#0;
   FC2_RECV_1[9] := B#16#0;
   FC2_RECV_1[10] := B#16#0;
   FC2_RECV_1[11] := B#16#0;
   FC2_RECV_1[12] := B#16#0;
   FC2_RECV_1[13] := B#16#0;
   FC2_RECV_1[14] := B#16#0;
   FC2_RECV_1[15] := B#16#0;
   FC2_RECV_1[16] := B#16#0;
   FC2_RECV_1[17] := B#16#0;
   FC2_RECV_1[18] := B#16#0;
   FC2_RECV_1[19] := B#16#0;
   FC2_RECV_1[20] := B#16#0;
   FC2_RECV_1[21] := B#16#0;
   FC2_RECV_1[22] := B#16#0;
   FC2_RECV_1[23] := B#16#0;
   FC2_RECV_1[24] := B#16#0;
   FC2_RECV_1[25] := B#16#0;
   FC2_RECV_1[26] := B#16#0;
   FC2_RECV_1[27] := B#16#0;
   FC2_RECV_1[28] := B#16#0;
   FC2_RECV_1[29] := B#16#0;
   FC2_RECV_1[30] := B#16#0;
   FC2_RECV_1[31] := B#16#0;
   FC2_RECV_1[32] := B#16#0;
   FC2_RECV_1[33] := B#16#0;
   FC2_RECV_1[34] := B#16#0;
   FC2_RECV_1[35] := B#16#0;
   FC2_RECV_1[36] := B#16#0;
   FC2_RECV_1[37] := B#16#0;
   FC2_RECV_1[38] := B#16#0;
   FC2_RECV_1[39] := B#16#0;
   FC2_RECV_1[40] := B#16#0;
   FC2_RECV_1[41] := B#16#0;
   FC2_RECV_1[42] := B#16#0;
   FC2_RECV_1[43] := B#16#0;
   FC2_RECV_1[44] := B#16#0;
   FC2_RECV_1[45] := B#16#0;
   FC2_RECV_1[46] := B#16#0;
   FC2_RECV_1[47] := B#16#0;
   FC2_RECV_1[48] := B#16#0;
   FC2_RECV_1[49] := B#16#0;
   FC2_RECV_1[50] := B#16#0;
   FC2_RECV_1[51] := B#16#0;
   FC2_RECV_1[52] := B#16#0;
   FC2_RECV_1[53] := B#16#0;
   FC2_RECV_1[54] := B#16#0;
   FC2_RECV_1[55] := B#16#0;
   FC2_RECV_1[56] := B#16#0;
   FC2_RECV_1[57] := B#16#0;
   FC2_RECV_1[58] := B#16#0;
   FC2_RECV_1[59] := B#16#0;
   FC2_RECV_1[60] := B#16#0;
   FC2_RECV_1[61] := B#16#0;
   FC2_RECV_1[62] := B#16#0;
   FC2_RECV_1[63] := B#16#0;
   FC2_RECV_1[64] := B#16#0;
   FC2_RECV_1[65] := B#16#0;
   FC2_RECV_1[66] := B#16#0;
   FC2_RECV_1[67] := B#16#0;
   FC2_RECV_1[68] := B#16#0;
   FC2_RECV_1[69] := B#16#0;
   FC2_RECV_1[70] := B#16#0;
   FC2_RECV_1[71] := B#16#0;
   FC2_RECV_1[72] := B#16#0;
   FC2_RECV_1[73] := B#16#0;
   FC2_RECV_1[74] := B#16#0;
   FC2_RECV_1[75] := B#16#0;
   FC2_RECV_1[76] := B#16#0;
   FC2_RECV_1[77] := B#16#0;
   FC2_RECV_1[78] := B#16#0;
   FC2_RECV_1[79] := B#16#0;
   FC2_RECV_1[80] := B#16#0;
   FC2_RECV_1[81] := B#16#0;
   FC2_RECV_1[82] := B#16#0;
   FC2_RECV_1[83] := B#16#0;
   FC2_RECV_1[84] := B#16#0;
   FC2_RECV_1[85] := B#16#0;
   FC2_RECV_1[86] := B#16#0;
   FC2_RECV_1[87] := B#16#0;
   FC2_RECV_1[88] := B#16#0;
   FC2_RECV_1[89] := B#16#0;
   FC2_RECV_1[90] := B#16#0;
   FC2_RECV_1[91] := B#16#0;
   FC2_RECV_1[92] := B#16#0;
   FC2_RECV_1[93] := B#16#0;
   FC2_RECV_1[94] := B#16#0;
   FC2_RECV_1[95] := B#16#0;
   FC2_RECV_1[96] := B#16#0;
   FC2_RECV_1[97] := B#16#0;
   FC2_RECV_1[98] := B#16#0;
   FC2_RECV_1[99] := B#16#0;
   FC2_RECV_1[100] := B#16#0;
   FC2_RECV_1[101] := B#16#0;
   FC2_RECV_1[102] := B#16#0;
   FC2_RECV_1[103] := B#16#0;
   FC2_RECV_1[104] := B#16#0;
   FC2_RECV_1[105] := B#16#0;
   FC2_RECV_1[106] := B#16#0;
   FC2_RECV_1[107] := B#16#0;
   FC2_RECV_1[108] := B#16#0;
   FC2_RECV_1[109] := B#16#0;
   FC2_RECV_1[110] := B#16#0;
   FC2_RECV_1[111] := B#16#0;
   FC2_RECV_1[112] := B#16#0;
   FC2_RECV_1[113] := B#16#0;
   FC2_RECV_1[114] := B#16#0;
   FC2_RECV_1[115] := B#16#0;
   FC2_RECV_1[116] := B#16#0;
   FC2_RECV_1[117] := B#16#0;
   FC2_RECV_1[118] := B#16#0;
   FC2_RECV_1[119] := B#16#0;
   FC2_RECV_1[120] := B#16#0;
   FC2_RECV_1[121] := B#16#0;
   FC2_RECV_1[122] := B#16#0;
   FC2_RECV_1[123] := B#16#0;
   FC2_RECV_1[124] := B#16#0;
   FC2_RECV_1[125] := B#16#0;
   FC2_RECV_1[126] := B#16#0;
   FC2_RECV_1[127] := B#16#0;
   FC2_RECV_1[128] := B#16#0;
   FC2_RECV_1[129] := B#16#0;
   FC2_RECV_1[130] := B#16#0;
   FC2_RECV_1[131] := B#16#0;
   FC2_RECV_1[132] := B#16#0;
   FC2_RECV_1[133] := B#16#0;
   FC2_RECV_1[134] := B#16#0;
   FC2_RECV_1[135] := B#16#0;
   FC2_RECV_1[136] := B#16#0;
   FC2_RECV_1[137] := B#16#0;
   FC2_RECV_1[138] := B#16#0;
   FC2_RECV_1[139] := B#16#0;
   FC2_RECV_1[140] := B#16#0;
   FC2_RECV_1[141] := B#16#0;
   FC2_RECV_1[142] := B#16#0;
   FC2_RECV_1[143] := B#16#0;
   FC2_RECV_1[144] := B#16#0;
   FC2_RECV_1[145] := B#16#0;
   FC2_RECV_1[146] := B#16#0;
   FC2_RECV_1[147] := B#16#0;
   FC2_RECV_1[148] := B#16#0;
   FC2_RECV_1[149] := B#16#0;
   FC2_RECV_1[150] := B#16#0;
   FC2_RECV_1[151] := B#16#0;
   FC2_RECV_1[152] := B#16#0;
   FC2_RECV_1[153] := B#16#0;
   FC2_RECV_1[154] := B#16#0;
   FC2_RECV_1[155] := B#16#0;
   FC2_RECV_1[156] := B#16#0;
   FC2_RECV_1[157] := B#16#0;
   FC2_RECV_1[158] := B#16#0;
   FC2_RECV_1[159] := B#16#0;
   FC2_RECV_1[160] := B#16#0;
   FC2_RECV_1[161] := B#16#0;
   FC2_RECV_1[162] := B#16#0;
   FC2_RECV_1[163] := B#16#0;
   FC2_RECV_1[164] := B#16#0;
   FC2_RECV_1[165] := B#16#0;
   FC2_RECV_1[166] := B#16#0;
   FC2_RECV_1[167] := B#16#0;
   FC2_RECV_1[168] := B#16#0;
   FC2_RECV_1[169] := B#16#0;
   FC2_RECV_1[170] := B#16#0;
   FC2_RECV_1[171] := B#16#0;
   FC2_RECV_1[172] := B#16#0;
   FC2_RECV_1[173] := B#16#0;
   FC2_RECV_1[174] := B#16#0;
   FC2_RECV_1[175] := B#16#0;
   FC2_RECV_1[176] := B#16#0;
   FC2_RECV_1[177] := B#16#0;
   FC2_RECV_1[178] := B#16#0;
   FC2_RECV_1[179] := B#16#0;
   FC2_RECV_1[180] := B#16#0;
   FC2_RECV_1[181] := B#16#0;
   FC2_RECV_1[182] := B#16#0;
   FC2_RECV_1[183] := B#16#0;
   FC2_RECV_1[184] := B#16#0;
   FC2_RECV_1[185] := B#16#0;
   FC2_RECV_1[186] := B#16#0;
   FC2_RECV_1[187] := B#16#0;
   FC2_RECV_1[188] := B#16#0;
   FC2_RECV_1[189] := B#16#0;
   FC2_RECV_1[190] := B#16#0;
   FC2_RECV_1[191] := B#16#0;
   FC2_RECV_1[192] := B#16#0;
   FC2_RECV_1[193] := B#16#0;
   FC2_RECV_1[194] := B#16#0;
   FC2_RECV_1[195] := B#16#0;
   FC2_RECV_1[196] := B#16#0;
   FC2_RECV_1[197] := B#16#0;
   FC2_RECV_1[198] := B#16#0;
   FC2_RECV_1[199] := B#16#0;
   FC2_RECV_1[200] := B#16#0;
   FC2_RECV_1[201] := B#16#0;
   FC2_RECV_1[202] := B#16#0;
   FC2_RECV_1[203] := B#16#0;
   FC2_RECV_1[204] := B#16#0;
   FC2_RECV_1[205] := B#16#0;
   FC2_RECV_1[206] := B#16#0;
   FC2_RECV_1[207] := B#16#0;
   FC2_RECV_1[208] := B#16#0;
   FC2_RECV_1[209] := B#16#0;
   FC2_RECV_1[210] := B#16#0;
   FC2_RECV_1[211] := B#16#0;
   FC2_RECV_1[212] := B#16#0;
   FC2_RECV_1[213] := B#16#0;
   FC2_RECV_1[214] := B#16#0;
   FC2_RECV_1[215] := B#16#0;
   FC2_RECV_1[216] := B#16#0;
   FC2_RECV_1[217] := B#16#0;
   FC2_RECV_1[218] := B#16#0;
   FC2_RECV_1[219] := B#16#0;
   FC2_RECV_1[220] := B#16#0;
   FC2_RECV_1[221] := B#16#0;
   FC2_RECV_1[222] := B#16#0;
   FC2_RECV_1[223] := B#16#0;
   FC2_RECV_1[224] := B#16#0;
   FC2_RECV_1[225] := B#16#0;
   FC2_RECV_1[226] := B#16#0;
   FC2_RECV_1[227] := B#16#0;
   FC2_RECV_1[228] := B#16#0;
   FC2_RECV_1[229] := B#16#0;
   FC2_RECV_1[230] := B#16#0;
   FC2_RECV_1[231] := B#16#0;
   FC2_RECV_1[232] := B#16#0;
   FC2_RECV_1[233] := B#16#0;
   FC2_RECV_1[234] := B#16#0;
   FC2_RECV_1[235] := B#16#0;
   FC2_RECV_1[236] := B#16#0;
   FC2_RECV_1[237] := B#16#0;
   FC2_RECV_1[238] := B#16#0;
   FC2_RECV_1[239] := B#16#0;
   FC2_RECV_1[240] := B#16#0;
   FC2_RECV_1[241] := B#16#0;
   FC2_RECV_1[242] := B#16#0;
   FC2_RECV_1[243] := B#16#0;
   FC2_RECV_1[244] := B#16#0;
   FC2_RECV_1[245] := B#16#0;
   FC2_RECV_1[246] := B#16#0;
   FC2_RECV_1[247] := B#16#0;
   FC2_RECV_1[248] := B#16#0;
   FC2_RECV_1[249] := B#16#0;
   FC2_RECV_1[250] := B#16#0;
   FC2_RECV_1[251] := B#16#0;
   FC2_RECV_1[252] := B#16#0;
   FC2_RECV_1[253] := B#16#0;
   FC2_RECV_1[254] := B#16#0;
   FC2_RECV_1[255] := B#16#0;
   FC2_RECV_1[256] := B#16#0;
   FC2_RECV_1[257] := B#16#0;
   FC2_RECV_1[258] := B#16#0;
   FC2_RECV_1[259] := B#16#0;
   FC2_RECV_1[260] := B#16#0;
   FC2_RECV_1[261] := B#16#0;
   FC2_RECV_1[262] := B#16#0;
   FC2_RECV_1[263] := B#16#0;
   FC2_RECV_1[264] := B#16#0;
   FC2_RECV_1[265] := B#16#0;
   FC2_RECV_1[266] := B#16#0;
   FC2_RECV_1[267] := B#16#0;
   FC2_RECV_1[268] := B#16#0;
   FC2_RECV_1[269] := B#16#0;
   FC2_RECV_1[270] := B#16#0;
   FC2_RECV_1[271] := B#16#0;
   FC2_RECV_1[272] := B#16#0;
   FC2_RECV_1[273] := B#16#0;
   FC2_RECV_1[274] := B#16#0;
   FC2_RECV_1[275] := B#16#0;
   FC2_RECV_1[276] := B#16#0;
   FC2_RECV_1[277] := B#16#0;
   FC2_RECV_1[278] := B#16#0;
   FC2_RECV_1[279] := B#16#0;
   FC2_RECV_1[280] := B#16#0;
   FC2_RECV_1[281] := B#16#0;
   FC2_RECV_1[282] := B#16#0;
   FC2_RECV_1[283] := B#16#0;
   FC2_RECV_1[284] := B#16#0;
   FC2_RECV_1[285] := B#16#0;
   FC2_RECV_1[286] := B#16#0;
   FC2_RECV_1[287] := B#16#0;
   FC2_RECV_1[288] := B#16#0;
   FC2_RECV_1[289] := B#16#0;
   FC2_RECV_1[290] := B#16#0;
   FC2_RECV_1[291] := B#16#0;
   FC2_RECV_1[292] := B#16#0;
   FC2_RECV_1[293] := B#16#0;
   FC2_RECV_1[294] := B#16#0;
   FC2_RECV_1[295] := B#16#0;
   FC2_RECV_1[296] := B#16#0;
   FC2_RECV_1[297] := B#16#0;
   FC2_RECV_1[298] := B#16#0;
   FC2_RECV_1[299] := B#16#0;
   FC2_RECV_1[300] := B#16#0;
   FC2_RECV_1[301] := B#16#0;
   FC2_RECV_1[302] := B#16#0;
   FC2_RECV_1[303] := B#16#0;
   FC2_RECV_1[304] := B#16#0;
   FC2_RECV_1[305] := B#16#0;
   FC2_RECV_1[306] := B#16#0;
   FC2_RECV_1[307] := B#16#0;
   FC2_RECV_1[308] := B#16#0;
   FC2_RECV_1[309] := B#16#0;
   FC2_RECV_1[310] := B#16#0;
   FC2_RECV_1[311] := B#16#0;
   FC2_RECV_1[312] := B#16#0;
   FC2_RECV_1[313] := B#16#0;
   FC2_RECV_1[314] := B#16#0;
   FC2_RECV_1[315] := B#16#0;
   FC2_RECV_1[316] := B#16#0;
   FC2_RECV_1[317] := B#16#0;
   FC2_RECV_1[318] := B#16#0;
   FC2_RECV_1[319] := B#16#0;
   FC2_RECV_1[320] := B#16#0;
   FC2_RECV_1[321] := B#16#0;
   FC2_RECV_1[322] := B#16#0;
   FC2_RECV_1[323] := B#16#0;
   FC2_RECV_1[324] := B#16#0;
   FC2_RECV_1[325] := B#16#0;
   FC2_RECV_1[326] := B#16#0;
   FC2_RECV_1[327] := B#16#0;
   FC2_RECV_1[328] := B#16#0;
   FC2_RECV_1[329] := B#16#0;
   FC2_RECV_1[330] := B#16#0;
   FC2_RECV_1[331] := B#16#0;
   FC2_RECV_1[332] := B#16#0;
   FC2_RECV_1[333] := B#16#0;
   FC2_RECV_1[334] := B#16#0;
   FC2_RECV_1[335] := B#16#0;
   FC2_RECV_1[336] := B#16#0;
   FC2_RECV_1[337] := B#16#0;
   FC2_RECV_1[338] := B#16#0;
   FC2_RECV_1[339] := B#16#0;
   FC2_RECV_1[340] := B#16#0;
   FC2_RECV_1[341] := B#16#0;
   FC2_RECV_1[342] := B#16#0;
   FC2_RECV_1[343] := B#16#0;
   FC2_RECV_1[344] := B#16#0;
   FC2_RECV_1[345] := B#16#0;
   FC2_RECV_1[346] := B#16#0;
   FC2_RECV_1[347] := B#16#0;
   FC2_RECV_1[348] := B#16#0;
   FC2_RECV_1[349] := B#16#0;
   FC2_RECV_1[350] := B#16#0;
   FC2_RECV_1[351] := B#16#0;
   FC2_RECV_1[352] := B#16#0;
   FC2_RECV_1[353] := B#16#0;
   FC2_RECV_1[354] := B#16#0;
   FC2_RECV_1[355] := B#16#0;
   FC2_RECV_1[356] := B#16#0;
   FC2_RECV_1[357] := B#16#0;
   FC2_RECV_1[358] := B#16#0;
   FC2_RECV_1[359] := B#16#0;
   FC2_RECV_1[360] := B#16#0;
   FC2_RECV_1[361] := B#16#0;
   FC2_RECV_1[362] := B#16#0;
   FC2_RECV_1[363] := B#16#0;
   FC2_RECV_1[364] := B#16#0;
   FC2_RECV_1[365] := B#16#0;
   FC2_RECV_1[366] := B#16#0;
   FC2_RECV_1[367] := B#16#0;
   FC2_RECV_1[368] := B#16#0;
   FC2_RECV_1[369] := B#16#0;
   FC2_RECV_1[370] := B#16#0;
   FC2_RECV_1[371] := B#16#0;
   FC2_RECV_1[372] := B#16#0;
   FC2_RECV_1[373] := B#16#0;
   FC2_RECV_1[374] := B#16#0;
   FC2_RECV_1[375] := B#16#0;
   FC2_RECV_1[376] := B#16#0;
   FC2_RECV_1[377] := B#16#0;
   FC2_RECV_1[378] := B#16#0;
   FC2_RECV_1[379] := B#16#0;
   FC2_RECV_1[380] := B#16#0;
   FC2_RECV_1[381] := B#16#0;
   FC2_RECV_1[382] := B#16#0;
   FC2_RECV_1[383] := B#16#0;
   FC2_RECV_1[384] := B#16#0;
   FC2_RECV_1[385] := B#16#0;
   FC2_RECV_1[386] := B#16#0;
   FC2_RECV_1[387] := B#16#0;
   FC2_RECV_1[388] := B#16#0;
   FC2_RECV_1[389] := B#16#0;
   FC2_RECV_1[390] := B#16#0;
   FC2_RECV_1[391] := B#16#0;
   FC2_RECV_1[392] := B#16#0;
   FC2_RECV_1[393] := B#16#0;
   FC2_RECV_1[394] := B#16#0;
   FC2_RECV_1[395] := B#16#0;
   FC2_RECV_1[396] := B#16#0;
   FC2_RECV_1[397] := B#16#0;
   FC2_RECV_1[398] := B#16#0;
   FC2_RECV_1[399] := B#16#0;
   FC2_RECV_1[400] := B#16#0;
   FC2_RECV_1[401] := B#16#0;
   FC2_RECV_1[402] := B#16#0;
   FC2_RECV_1[403] := B#16#0;
   FC2_RECV_1[404] := B#16#0;
   FC2_RECV_1[405] := B#16#0;
   FC2_RECV_1[406] := B#16#0;
   FC2_RECV_1[407] := B#16#0;
   FC2_RECV_1[408] := B#16#0;
   FC2_RECV_1[409] := B#16#0;
   FC2_RECV_1[410] := B#16#0;
   FC2_RECV_1[411] := B#16#0;
   FC2_RECV_1[412] := B#16#0;
   FC2_RECV_1[413] := B#16#0;
   FC2_RECV_1[414] := B#16#0;
   FC2_RECV_1[415] := B#16#0;
   FC2_RECV_1[416] := B#16#0;
   FC2_RECV_1[417] := B#16#0;
   FC2_RECV_1[418] := B#16#0;
   FC2_RECV_1[419] := B#16#0;
   FC2_RECV_1[420] := B#16#0;
   FC2_RECV_1[421] := B#16#0;
   FC2_RECV_1[422] := B#16#0;
   FC2_RECV_1[423] := B#16#0;
   FC2_RECV_1[424] := B#16#0;
   FC2_RECV_1[425] := B#16#0;
   FC2_RECV_1[426] := B#16#0;
   FC2_RECV_1[427] := B#16#0;
   FC2_RECV_1[428] := B#16#0;
   FC2_RECV_1[429] := B#16#0;
   FC2_RECV_1[430] := B#16#0;
   FC2_RECV_1[431] := B#16#0;
   FC2_RECV_1[432] := B#16#0;
   FC2_RECV_1[433] := B#16#0;
   FC2_RECV_1[434] := B#16#0;
   FC2_RECV_1[435] := B#16#0;
   FC2_RECV_1[436] := B#16#0;
   FC2_RECV_1[437] := B#16#0;
   FC2_RECV_1[438] := B#16#0;
   FC2_RECV_1[439] := B#16#0;
   FC2_RECV_1[440] := B#16#0;
   FC2_RECV_1[441] := B#16#0;
   FC2_RECV_1[442] := B#16#0;
   FC2_RECV_1[443] := B#16#0;
   FC2_RECV_1[444] := B#16#0;
   FC2_RECV_1[445] := B#16#0;
   FC2_RECV_1[446] := B#16#0;
   FC2_RECV_1[447] := B#16#0;
   FC2_RECV_1[448] := B#16#0;
   FC2_RECV_1[449] := B#16#0;
   FC2_RECV_1[450] := B#16#0;
   FC2_RECV_1[451] := B#16#0;
   FC2_RECV_1[452] := B#16#0;
   FC2_RECV_1[453] := B#16#0;
   FC2_RECV_1[454] := B#16#0;
   FC2_RECV_1[455] := B#16#0;
   FC2_RECV_1[456] := B#16#0;
   FC2_RECV_1[457] := B#16#0;
   FC2_RECV_1[458] := B#16#0;
   FC2_RECV_1[459] := B#16#0;
   FC2_RECV_1[460] := B#16#0;
   FC2_RECV_1[461] := B#16#0;
   FC2_RECV_1[462] := B#16#0;
   FC2_RECV_1[463] := B#16#0;
   FC2_RECV_1[464] := B#16#0;
   FC2_RECV_1[465] := B#16#0;
   FC2_RECV_1[466] := B#16#0;
   FC2_RECV_1[467] := B#16#0;
   FC2_RECV_1[468] := B#16#0;
   FC2_RECV_1[469] := B#16#0;
   FC2_RECV_1[470] := B#16#0;
   FC2_RECV_1[471] := B#16#0;
   FC2_RECV_1[472] := B#16#0;
   FC2_RECV_1[473] := B#16#0;
   FC2_RECV_1[474] := B#16#0;
   FC2_RECV_1[475] := B#16#0;
   FC2_RECV_1[476] := B#16#0;
   FC2_RECV_1[477] := B#16#0;
   FC2_RECV_1[478] := B#16#0;
   FC2_RECV_1[479] := B#16#0;
   FC2_RECV_1[480] := B#16#0;
   FC2_RECV_1[481] := B#16#0;
   FC2_RECV_1[482] := B#16#0;
   FC2_RECV_1[483] := B#16#0;
   FC2_RECV_1[484] := B#16#0;
   FC2_RECV_1[485] := B#16#0;
   FC2_RECV_1[486] := B#16#0;
   FC2_RECV_1[487] := B#16#0;
   FC2_RECV_1[488] := B#16#0;
   FC2_RECV_1[489] := B#16#0;
   FC2_RECV_1[490] := B#16#0;
   FC2_RECV_1[491] := B#16#0;
   FC2_RECV_1[492] := B#16#0;
   FC2_RECV_1[493] := B#16#0;
   FC2_RECV_1[494] := B#16#0;
   FC2_RECV_1[495] := B#16#0;
   FC2_RECV_1[496] := B#16#0;
   FC2_RECV_1[497] := B#16#0;
   FC2_RECV_1[498] := B#16#0;
   FC2_RECV_1[499] := B#16#0;
   FC2_RECV_1[500] := B#16#0;
   FC2_RECV_1[501] := B#16#0;
   FC2_RECV_1[502] := B#16#0;
   FC2_RECV_1[503] := B#16#0;
   FC2_RECV_1[504] := B#16#0;
   FC2_RECV_1[505] := B#16#0;
   FC2_RECV_1[506] := B#16#0;
   FC2_RECV_1[507] := B#16#0;
   FC2_RECV_1[508] := B#16#0;
   FC2_RECV_1[509] := B#16#0;
   FC2_RECV_1[510] := B#16#0;
   FC2_RECV_1[511] := B#16#0;
   FC2_RECV_1[512] := B#16#0;
   FC2_RECV_1[513] := B#16#0;
   FC2_RECV_1[514] := B#16#0;
   FC2_RECV_1[515] := B#16#0;
   FC2_RECV_1[516] := B#16#0;
   FC2_RECV_1[517] := B#16#0;
   FC2_RECV_1[518] := B#16#0;
   FC2_RECV_1[519] := B#16#0;
   FC2_RECV_1[520] := B#16#0;
   FC2_RECV_1[521] := B#16#0;
   FC2_RECV_1[522] := B#16#0;
   FC2_RECV_1[523] := B#16#0;
   FC2_RECV_1[524] := B#16#0;
   FC2_RECV_1[525] := B#16#0;
   FC2_RECV_1[526] := B#16#0;
   FC2_RECV_1[527] := B#16#0;
   FC2_RECV_1[528] := B#16#0;
   FC2_RECV_1[529] := B#16#0;
   FC2_RECV_1[530] := B#16#0;
   FC2_RECV_1[531] := B#16#0;
   FC2_RECV_1[532] := B#16#0;
   FC2_RECV_1[533] := B#16#0;
   FC2_RECV_1[534] := B#16#0;
   FC2_RECV_1[535] := B#16#0;
   FC2_RECV_1[536] := B#16#0;
   FC2_RECV_1[537] := B#16#0;
   FC2_RECV_1[538] := B#16#0;
   FC2_RECV_1[539] := B#16#0;
   FC2_RECV_1[540] := B#16#0;
   FC2_RECV_1[541] := B#16#0;
   FC2_RECV_1[542] := B#16#0;
   FC2_RECV_1[543] := B#16#0;
   FC2_RECV_1[544] := B#16#0;
   FC2_RECV_1[545] := B#16#0;
   FC2_RECV_1[546] := B#16#0;
   FC2_RECV_1[547] := B#16#0;
   FC2_RECV_1[548] := B#16#0;
   FC2_RECV_1[549] := B#16#0;
   FC2_RECV_1[550] := B#16#0;
   FC2_RECV_1[551] := B#16#0;
   FC2_RECV_1[552] := B#16#0;
   FC2_RECV_1[553] := B#16#0;
   FC2_RECV_1[554] := B#16#0;
   FC2_RECV_1[555] := B#16#0;
   FC2_RECV_1[556] := B#16#0;
   FC2_RECV_1[557] := B#16#0;
   FC2_RECV_1[558] := B#16#0;
   FC2_RECV_1[559] := B#16#0;
   FC2_RECV_1[560] := B#16#0;
   FC2_RECV_1[561] := B#16#0;
   FC2_RECV_1[562] := B#16#0;
   FC2_RECV_1[563] := B#16#0;
   FC2_RECV_1[564] := B#16#0;
   FC2_RECV_1[565] := B#16#0;
   FC2_RECV_1[566] := B#16#0;
   FC2_RECV_1[567] := B#16#0;
   FC2_RECV_1[568] := B#16#0;
   FC2_RECV_1[569] := B#16#0;
   FC2_RECV_1[570] := B#16#0;
   FC2_RECV_1[571] := B#16#0;
   FC2_RECV_1[572] := B#16#0;
   FC2_RECV_1[573] := B#16#0;
   FC2_RECV_1[574] := B#16#0;
   FC2_RECV_1[575] := B#16#0;
   FC2_RECV_1[576] := B#16#0;
   FC2_RECV_1[577] := B#16#0;
   FC2_RECV_1[578] := B#16#0;
   FC2_RECV_1[579] := B#16#0;
   FC2_RECV_1[580] := B#16#0;
   FC2_RECV_1[581] := B#16#0;
   FC2_RECV_1[582] := B#16#0;
   FC2_RECV_1[583] := B#16#0;
   FC2_RECV_1[584] := B#16#0;
   FC2_RECV_1[585] := B#16#0;
   FC2_RECV_1[586] := B#16#0;
   FC2_RECV_1[587] := B#16#0;
   FC2_RECV_1[588] := B#16#0;
   FC2_RECV_1[589] := B#16#0;
   FC2_RECV_1[590] := B#16#0;
   FC2_RECV_1[591] := B#16#0;
   FC2_RECV_1[592] := B#16#0;
   FC2_RECV_1[593] := B#16#0;
   FC2_RECV_1[594] := B#16#0;
   FC2_RECV_1[595] := B#16#0;
   FC2_RECV_1[596] := B#16#0;
   FC2_RECV_1[597] := B#16#0;
   FC2_RECV_1[598] := B#16#0;
   FC2_RECV_1[599] := B#16#0;
   FC2_RECV_1[600] := B#16#0;
   FC2_RECV_1[601] := B#16#0;
   FC2_RECV_1[602] := B#16#0;
   FC2_RECV_1[603] := B#16#0;
   FC2_RECV_1[604] := B#16#0;
   FC2_RECV_1[605] := B#16#0;
   FC2_RECV_1[606] := B#16#0;
   FC2_RECV_1[607] := B#16#0;
   FC2_RECV_1[608] := B#16#0;
   FC2_RECV_1[609] := B#16#0;
   FC2_RECV_1[610] := B#16#0;
   FC2_RECV_1[611] := B#16#0;
   FC2_RECV_1[612] := B#16#0;
   FC2_RECV_1[613] := B#16#0;
   FC2_RECV_1[614] := B#16#0;
   FC2_RECV_1[615] := B#16#0;
   FC2_RECV_1[616] := B#16#0;
   FC2_RECV_1[617] := B#16#0;
   FC2_RECV_1[618] := B#16#0;
   FC2_RECV_1[619] := B#16#0;
   FC2_RECV_1[620] := B#16#0;
   FC2_RECV_1[621] := B#16#0;
   FC2_RECV_1[622] := B#16#0;
   FC2_RECV_1[623] := B#16#0;
   FC2_RECV_1[624] := B#16#0;
   FC2_RECV_1[625] := B#16#0;
   FC2_RECV_1[626] := B#16#0;
   FC2_RECV_1[627] := B#16#0;
   FC2_RECV_1[628] := B#16#0;
   FC2_RECV_1[629] := B#16#0;
   FC2_RECV_1[630] := B#16#0;
   FC2_RECV_1[631] := B#16#0;
   FC2_RECV_1[632] := B#16#0;
   FC2_RECV_1[633] := B#16#0;
   FC2_RECV_1[634] := B#16#0;
   FC2_RECV_1[635] := B#16#0;
   FC2_RECV_1[636] := B#16#0;
   FC2_RECV_1[637] := B#16#0;
   FC2_RECV_1[638] := B#16#0;
   FC2_RECV_1[639] := B#16#0;
   FC2_RECV_1[640] := B#16#0;
   FC2_RECV_1[641] := B#16#0;
   FC2_RECV_1[642] := B#16#0;
   FC2_RECV_1[643] := B#16#0;
   FC2_RECV_1[644] := B#16#0;
   FC2_RECV_1[645] := B#16#0;
   FC2_RECV_1[646] := B#16#0;
   FC2_RECV_1[647] := B#16#0;
   FC2_RECV_1[648] := B#16#0;
   FC2_RECV_1[649] := B#16#0;
   FC2_RECV_1[650] := B#16#0;
   FC2_RECV_1[651] := B#16#0;
   FC2_RECV_1[652] := B#16#0;
   FC2_RECV_1[653] := B#16#0;
   FC2_RECV_1[654] := B#16#0;
   FC2_RECV_1[655] := B#16#0;
   FC2_RECV_1[656] := B#16#0;
   FC2_RECV_1[657] := B#16#0;
   FC2_RECV_1[658] := B#16#0;
   FC2_RECV_1[659] := B#16#0;
   FC2_RECV_1[660] := B#16#0;
   FC2_RECV_1[661] := B#16#0;
   FC2_RECV_1[662] := B#16#0;
   FC2_RECV_1[663] := B#16#0;
   FC2_RECV_1[664] := B#16#0;
   FC2_RECV_1[665] := B#16#0;
   FC2_RECV_1[666] := B#16#0;
   FC2_RECV_1[667] := B#16#0;
   FC2_RECV_1[668] := B#16#0;
   FC2_RECV_1[669] := B#16#0;
   FC2_RECV_1[670] := B#16#0;
   FC2_RECV_1[671] := B#16#0;
   FC2_RECV_1[672] := B#16#0;
   FC2_RECV_1[673] := B#16#0;
   FC2_RECV_1[674] := B#16#0;
   FC2_RECV_1[675] := B#16#0;
   FC2_RECV_1[676] := B#16#0;
   FC2_RECV_1[677] := B#16#0;
   FC2_RECV_1[678] := B#16#0;
   FC2_RECV_1[679] := B#16#0;
   FC2_RECV_1[680] := B#16#0;
   FC2_RECV_1[681] := B#16#0;
   FC2_RECV_1[682] := B#16#0;
   FC2_RECV_1[683] := B#16#0;
   FC2_RECV_1[684] := B#16#0;
   FC2_RECV_1[685] := B#16#0;
   FC2_RECV_1[686] := B#16#0;
   FC2_RECV_1[687] := B#16#0;
   FC2_RECV_1[688] := B#16#0;
   FC2_RECV_1[689] := B#16#0;
   FC2_RECV_1[690] := B#16#0;
   FC2_RECV_1[691] := B#16#0;
   FC2_RECV_1[692] := B#16#0;
   FC2_RECV_1[693] := B#16#0;
   FC2_RECV_1[694] := B#16#0;
   FC2_RECV_1[695] := B#16#0;
   FC2_RECV_1[696] := B#16#0;
   FC2_RECV_1[697] := B#16#0;
   FC2_RECV_1[698] := B#16#0;
   FC2_RECV_1[699] := B#16#0;
END_DATA_BLOCK

DATA_BLOCK DB 325
TITLE =
VERSION : 0.1


  STRUCT
   DP_DIAG1 : ARRAY  [1 .. 100 ] OF BYTE ;
   DP_DIAG2 : ARRAY  [1 .. 100 ] OF BYTE ;
   DP_DIAG3 : ARRAY  [1 .. 100 ] OF BYTE ;
   DP_DIAG4 : ARRAY  [1 .. 100 ] OF BYTE ;
   DP_DIAG5 : ARRAY  [1 .. 100 ] OF BYTE ;
   DP_DIAG6 : ARRAY  [1 .. 100 ] OF BYTE ;
   DP_DIAG7 : ARRAY  [1 .. 100 ] OF BYTE ;
   DP_DIAG8 : ARRAY  [1 .. 100 ] OF BYTE ;
   DP_DIAG9 : ARRAY  [1 .. 100 ] OF BYTE ;
   DP_DIAG10 : ARRAY  [1 .. 100 ] OF BYTE ;
  END_STRUCT ;
BEGIN
   DP_DIAG1[1] := B#16#0;
   DP_DIAG1[2] := B#16#0;
   DP_DIAG1[3] := B#16#0;
   DP_DIAG1[4] := B#16#0;
   DP_DIAG1[5] := B#16#0;
   DP_DIAG1[6] := B#16#0;
   DP_DIAG1[7] := B#16#0;
   DP_DIAG1[8] := B#16#0;
   DP_DIAG1[9] := B#16#0;
   DP_DIAG1[10] := B#16#0;
   DP_DIAG1[11] := B#16#0;
   DP_DIAG1[12] := B#16#0;
   DP_DIAG1[13] := B#16#0;
   DP_DIAG1[14] := B#16#0;
   DP_DIAG1[15] := B#16#0;
   DP_DIAG1[16] := B#16#0;
   DP_DIAG1[17] := B#16#0;
   DP_DIAG1[18] := B#16#0;
   DP_DIAG1[19] := B#16#0;
   DP_DIAG1[20] := B#16#0;
   DP_DIAG1[21] := B#16#0;
   DP_DIAG1[22] := B#16#0;
   DP_DIAG1[23] := B#16#0;
   DP_DIAG1[24] := B#16#0;
   DP_DIAG1[25] := B#16#0;
   DP_DIAG1[26] := B#16#0;
   DP_DIAG1[27] := B#16#0;
   DP_DIAG1[28] := B#16#0;
   DP_DIAG1[29] := B#16#0;
   DP_DIAG1[30] := B#16#0;
   DP_DIAG1[31] := B#16#0;
   DP_DIAG1[32] := B#16#0;
   DP_DIAG1[33] := B#16#0;
   DP_DIAG1[34] := B#16#0;
   DP_DIAG1[35] := B#16#0;
   DP_DIAG1[36] := B#16#0;
   DP_DIAG1[37] := B#16#0;
   DP_DIAG1[38] := B#16#0;
   DP_DIAG1[39] := B#16#0;
   DP_DIAG1[40] := B#16#0;
   DP_DIAG1[41] := B#16#0;
   DP_DIAG1[42] := B#16#0;
   DP_DIAG1[43] := B#16#0;
   DP_DIAG1[44] := B#16#0;
   DP_DIAG1[45] := B#16#0;
   DP_DIAG1[46] := B#16#0;
   DP_DIAG1[47] := B#16#0;
   DP_DIAG1[48] := B#16#0;
   DP_DIAG1[49] := B#16#0;
   DP_DIAG1[50] := B#16#0;
   DP_DIAG1[51] := B#16#0;
   DP_DIAG1[52] := B#16#0;
   DP_DIAG1[53] := B#16#0;
   DP_DIAG1[54] := B#16#0;
   DP_DIAG1[55] := B#16#0;
   DP_DIAG1[56] := B#16#0;
   DP_DIAG1[57] := B#16#0;
   DP_DIAG1[58] := B#16#0;
   DP_DIAG1[59] := B#16#0;
   DP_DIAG1[60] := B#16#0;
   DP_DIAG1[61] := B#16#0;
   DP_DIAG1[62] := B#16#0;
   DP_DIAG1[63] := B#16#0;
   DP_DIAG1[64] := B#16#0;
   DP_DIAG1[65] := B#16#0;
   DP_DIAG1[66] := B#16#0;
   DP_DIAG1[67] := B#16#0;
   DP_DIAG1[68] := B#16#0;
   DP_DIAG1[69] := B#16#0;
   DP_DIAG1[70] := B#16#0;
   DP_DIAG1[71] := B#16#0;
   DP_DIAG1[72] := B#16#0;
   DP_DIAG1[73] := B#16#0;
   DP_DIAG1[74] := B#16#0;
   DP_DIAG1[75] := B#16#0;
   DP_DIAG1[76] := B#16#0;
   DP_DIAG1[77] := B#16#0;
   DP_DIAG1[78] := B#16#0;
   DP_DIAG1[79] := B#16#0;
   DP_DIAG1[80] := B#16#0;
   DP_DIAG1[81] := B#16#0;
   DP_DIAG1[82] := B#16#0;
   DP_DIAG1[83] := B#16#0;
   DP_DIAG1[84] := B#16#0;
   DP_DIAG1[85] := B#16#0;
   DP_DIAG1[86] := B#16#0;
   DP_DIAG1[87] := B#16#0;
   DP_DIAG1[88] := B#16#0;
   DP_DIAG1[89] := B#16#0;
   DP_DIAG1[90] := B#16#0;
   DP_DIAG1[91] := B#16#0;
   DP_DIAG1[92] := B#16#0;
   DP_DIAG1[93] := B#16#0;
   DP_DIAG1[94] := B#16#0;
   DP_DIAG1[95] := B#16#0;
   DP_DIAG1[96] := B#16#0;
   DP_DIAG1[97] := B#16#0;
   DP_DIAG1[98] := B#16#0;
   DP_DIAG1[99] := B#16#0;
   DP_DIAG1[100] := B#16#0;
   DP_DIAG2[1] := B#16#0;
   DP_DIAG2[2] := B#16#0;
   DP_DIAG2[3] := B#16#0;
   DP_DIAG2[4] := B#16#0;
   DP_DIAG2[5] := B#16#0;
   DP_DIAG2[6] := B#16#0;
   DP_DIAG2[7] := B#16#0;
   DP_DIAG2[8] := B#16#0;
   DP_DIAG2[9] := B#16#0;
   DP_DIAG2[10] := B#16#0;
   DP_DIAG2[11] := B#16#0;
   DP_DIAG2[12] := B#16#0;
   DP_DIAG2[13] := B#16#0;
   DP_DIAG2[14] := B#16#0;
   DP_DIAG2[15] := B#16#0;
   DP_DIAG2[16] := B#16#0;
   DP_DIAG2[17] := B#16#0;
   DP_DIAG2[18] := B#16#0;
   DP_DIAG2[19] := B#16#0;
   DP_DIAG2[20] := B#16#0;
   DP_DIAG2[21] := B#16#0;
   DP_DIAG2[22] := B#16#0;
   DP_DIAG2[23] := B#16#0;
   DP_DIAG2[24] := B#16#0;
   DP_DIAG2[25] := B#16#0;
   DP_DIAG2[26] := B#16#0;
   DP_DIAG2[27] := B#16#0;
   DP_DIAG2[28] := B#16#0;
   DP_DIAG2[29] := B#16#0;
   DP_DIAG2[30] := B#16#0;
   DP_DIAG2[31] := B#16#0;
   DP_DIAG2[32] := B#16#0;
   DP_DIAG2[33] := B#16#0;
   DP_DIAG2[34] := B#16#0;
   DP_DIAG2[35] := B#16#0;
   DP_DIAG2[36] := B#16#0;
   DP_DIAG2[37] := B#16#0;
   DP_DIAG2[38] := B#16#0;
   DP_DIAG2[39] := B#16#0;
   DP_DIAG2[40] := B#16#0;
   DP_DIAG2[41] := B#16#0;
   DP_DIAG2[42] := B#16#0;
   DP_DIAG2[43] := B#16#0;
   DP_DIAG2[44] := B#16#0;
   DP_DIAG2[45] := B#16#0;
   DP_DIAG2[46] := B#16#0;
   DP_DIAG2[47] := B#16#0;
   DP_DIAG2[48] := B#16#0;
   DP_DIAG2[49] := B#16#0;
   DP_DIAG2[50] := B#16#0;
   DP_DIAG2[51] := B#16#0;
   DP_DIAG2[52] := B#16#0;
   DP_DIAG2[53] := B#16#0;
   DP_DIAG2[54] := B#16#0;
   DP_DIAG2[55] := B#16#0;
   DP_DIAG2[56] := B#16#0;
   DP_DIAG2[57] := B#16#0;
   DP_DIAG2[58] := B#16#0;
   DP_DIAG2[59] := B#16#0;
   DP_DIAG2[60] := B#16#0;
   DP_DIAG2[61] := B#16#0;
   DP_DIAG2[62] := B#16#0;
   DP_DIAG2[63] := B#16#0;
   DP_DIAG2[64] := B#16#0;
   DP_DIAG2[65] := B#16#0;
   DP_DIAG2[66] := B#16#0;
   DP_DIAG2[67] := B#16#0;
   DP_DIAG2[68] := B#16#0;
   DP_DIAG2[69] := B#16#0;
   DP_DIAG2[70] := B#16#0;
   DP_DIAG2[71] := B#16#0;
   DP_DIAG2[72] := B#16#0;
   DP_DIAG2[73] := B#16#0;
   DP_DIAG2[74] := B#16#0;
   DP_DIAG2[75] := B#16#0;
   DP_DIAG2[76] := B#16#0;
   DP_DIAG2[77] := B#16#0;
   DP_DIAG2[78] := B#16#0;
   DP_DIAG2[79] := B#16#0;
   DP_DIAG2[80] := B#16#0;
   DP_DIAG2[81] := B#16#0;
   DP_DIAG2[82] := B#16#0;
   DP_DIAG2[83] := B#16#0;
   DP_DIAG2[84] := B#16#0;
   DP_DIAG2[85] := B#16#0;
   DP_DIAG2[86] := B#16#0;
   DP_DIAG2[87] := B#16#0;
   DP_DIAG2[88] := B#16#0;
   DP_DIAG2[89] := B#16#0;
   DP_DIAG2[90] := B#16#0;
   DP_DIAG2[91] := B#16#0;
   DP_DIAG2[92] := B#16#0;
   DP_DIAG2[93] := B#16#0;
   DP_DIAG2[94] := B#16#0;
   DP_DIAG2[95] := B#16#0;
   DP_DIAG2[96] := B#16#0;
   DP_DIAG2[97] := B#16#0;
   DP_DIAG2[98] := B#16#0;
   DP_DIAG2[99] := B#16#0;
   DP_DIAG2[100] := B#16#0;
   DP_DIAG3[1] := B#16#0;
   DP_DIAG3[2] := B#16#0;
   DP_DIAG3[3] := B#16#0;
   DP_DIAG3[4] := B#16#0;
   DP_DIAG3[5] := B#16#0;
   DP_DIAG3[6] := B#16#0;
   DP_DIAG3[7] := B#16#0;
   DP_DIAG3[8] := B#16#0;
   DP_DIAG3[9] := B#16#0;
   DP_DIAG3[10] := B#16#0;
   DP_DIAG3[11] := B#16#0;
   DP_DIAG3[12] := B#16#0;
   DP_DIAG3[13] := B#16#0;
   DP_DIAG3[14] := B#16#0;
   DP_DIAG3[15] := B#16#0;
   DP_DIAG3[16] := B#16#0;
   DP_DIAG3[17] := B#16#0;
   DP_DIAG3[18] := B#16#0;
   DP_DIAG3[19] := B#16#0;
   DP_DIAG3[20] := B#16#0;
   DP_DIAG3[21] := B#16#0;
   DP_DIAG3[22] := B#16#0;
   DP_DIAG3[23] := B#16#0;
   DP_DIAG3[24] := B#16#0;
   DP_DIAG3[25] := B#16#0;
   DP_DIAG3[26] := B#16#0;
   DP_DIAG3[27] := B#16#0;
   DP_DIAG3[28] := B#16#0;
   DP_DIAG3[29] := B#16#0;
   DP_DIAG3[30] := B#16#0;
   DP_DIAG3[31] := B#16#0;
   DP_DIAG3[32] := B#16#0;
   DP_DIAG3[33] := B#16#0;
   DP_DIAG3[34] := B#16#0;
   DP_DIAG3[35] := B#16#0;
   DP_DIAG3[36] := B#16#0;
   DP_DIAG3[37] := B#16#0;
   DP_DIAG3[38] := B#16#0;
   DP_DIAG3[39] := B#16#0;
   DP_DIAG3[40] := B#16#0;
   DP_DIAG3[41] := B#16#0;
   DP_DIAG3[42] := B#16#0;
   DP_DIAG3[43] := B#16#0;
   DP_DIAG3[44] := B#16#0;
   DP_DIAG3[45] := B#16#0;
   DP_DIAG3[46] := B#16#0;
   DP_DIAG3[47] := B#16#0;
   DP_DIAG3[48] := B#16#0;
   DP_DIAG3[49] := B#16#0;
   DP_DIAG3[50] := B#16#0;
   DP_DIAG3[51] := B#16#0;
   DP_DIAG3[52] := B#16#0;
   DP_DIAG3[53] := B#16#0;
   DP_DIAG3[54] := B#16#0;
   DP_DIAG3[55] := B#16#0;
   DP_DIAG3[56] := B#16#0;
   DP_DIAG3[57] := B#16#0;
   DP_DIAG3[58] := B#16#0;
   DP_DIAG3[59] := B#16#0;
   DP_DIAG3[60] := B#16#0;
   DP_DIAG3[61] := B#16#0;
   DP_DIAG3[62] := B#16#0;
   DP_DIAG3[63] := B#16#0;
   DP_DIAG3[64] := B#16#0;
   DP_DIAG3[65] := B#16#0;
   DP_DIAG3[66] := B#16#0;
   DP_DIAG3[67] := B#16#0;
   DP_DIAG3[68] := B#16#0;
   DP_DIAG3[69] := B#16#0;
   DP_DIAG3[70] := B#16#0;
   DP_DIAG3[71] := B#16#0;
   DP_DIAG3[72] := B#16#0;
   DP_DIAG3[73] := B#16#0;
   DP_DIAG3[74] := B#16#0;
   DP_DIAG3[75] := B#16#0;
   DP_DIAG3[76] := B#16#0;
   DP_DIAG3[77] := B#16#0;
   DP_DIAG3[78] := B#16#0;
   DP_DIAG3[79] := B#16#0;
   DP_DIAG3[80] := B#16#0;
   DP_DIAG3[81] := B#16#0;
   DP_DIAG3[82] := B#16#0;
   DP_DIAG3[83] := B#16#0;
   DP_DIAG3[84] := B#16#0;
   DP_DIAG3[85] := B#16#0;
   DP_DIAG3[86] := B#16#0;
   DP_DIAG3[87] := B#16#0;
   DP_DIAG3[88] := B#16#0;
   DP_DIAG3[89] := B#16#0;
   DP_DIAG3[90] := B#16#0;
   DP_DIAG3[91] := B#16#0;
   DP_DIAG3[92] := B#16#0;
   DP_DIAG3[93] := B#16#0;
   DP_DIAG3[94] := B#16#0;
   DP_DIAG3[95] := B#16#0;
   DP_DIAG3[96] := B#16#0;
   DP_DIAG3[97] := B#16#0;
   DP_DIAG3[98] := B#16#0;
   DP_DIAG3[99] := B#16#0;
   DP_DIAG3[100] := B#16#0;
   DP_DIAG4[1] := B#16#0;
   DP_DIAG4[2] := B#16#0;
   DP_DIAG4[3] := B#16#0;
   DP_DIAG4[4] := B#16#0;
   DP_DIAG4[5] := B#16#0;
   DP_DIAG4[6] := B#16#0;
   DP_DIAG4[7] := B#16#0;
   DP_DIAG4[8] := B#16#0;
   DP_DIAG4[9] := B#16#0;
   DP_DIAG4[10] := B#16#0;
   DP_DIAG4[11] := B#16#0;
   DP_DIAG4[12] := B#16#0;
   DP_DIAG4[13] := B#16#0;
   DP_DIAG4[14] := B#16#0;
   DP_DIAG4[15] := B#16#0;
   DP_DIAG4[16] := B#16#0;
   DP_DIAG4[17] := B#16#0;
   DP_DIAG4[18] := B#16#0;
   DP_DIAG4[19] := B#16#0;
   DP_DIAG4[20] := B#16#0;
   DP_DIAG4[21] := B#16#0;
   DP_DIAG4[22] := B#16#0;
   DP_DIAG4[23] := B#16#0;
   DP_DIAG4[24] := B#16#0;
   DP_DIAG4[25] := B#16#0;
   DP_DIAG4[26] := B#16#0;
   DP_DIAG4[27] := B#16#0;
   DP_DIAG4[28] := B#16#0;
   DP_DIAG4[29] := B#16#0;
   DP_DIAG4[30] := B#16#0;
   DP_DIAG4[31] := B#16#0;
   DP_DIAG4[32] := B#16#0;
   DP_DIAG4[33] := B#16#0;
   DP_DIAG4[34] := B#16#0;
   DP_DIAG4[35] := B#16#0;
   DP_DIAG4[36] := B#16#0;
   DP_DIAG4[37] := B#16#0;
   DP_DIAG4[38] := B#16#0;
   DP_DIAG4[39] := B#16#0;
   DP_DIAG4[40] := B#16#0;
   DP_DIAG4[41] := B#16#0;
   DP_DIAG4[42] := B#16#0;
   DP_DIAG4[43] := B#16#0;
   DP_DIAG4[44] := B#16#0;
   DP_DIAG4[45] := B#16#0;
   DP_DIAG4[46] := B#16#0;
   DP_DIAG4[47] := B#16#0;
   DP_DIAG4[48] := B#16#0;
   DP_DIAG4[49] := B#16#0;
   DP_DIAG4[50] := B#16#0;
   DP_DIAG4[51] := B#16#0;
   DP_DIAG4[52] := B#16#0;
   DP_DIAG4[53] := B#16#0;
   DP_DIAG4[54] := B#16#0;
   DP_DIAG4[55] := B#16#0;
   DP_DIAG4[56] := B#16#0;
   DP_DIAG4[57] := B#16#0;
   DP_DIAG4[58] := B#16#0;
   DP_DIAG4[59] := B#16#0;
   DP_DIAG4[60] := B#16#0;
   DP_DIAG4[61] := B#16#0;
   DP_DIAG4[62] := B#16#0;
   DP_DIAG4[63] := B#16#0;
   DP_DIAG4[64] := B#16#0;
   DP_DIAG4[65] := B#16#0;
   DP_DIAG4[66] := B#16#0;
   DP_DIAG4[67] := B#16#0;
   DP_DIAG4[68] := B#16#0;
   DP_DIAG4[69] := B#16#0;
   DP_DIAG4[70] := B#16#0;
   DP_DIAG4[71] := B#16#0;
   DP_DIAG4[72] := B#16#0;
   DP_DIAG4[73] := B#16#0;
   DP_DIAG4[74] := B#16#0;
   DP_DIAG4[75] := B#16#0;
   DP_DIAG4[76] := B#16#0;
   DP_DIAG4[77] := B#16#0;
   DP_DIAG4[78] := B#16#0;
   DP_DIAG4[79] := B#16#0;
   DP_DIAG4[80] := B#16#0;
   DP_DIAG4[81] := B#16#0;
   DP_DIAG4[82] := B#16#0;
   DP_DIAG4[83] := B#16#0;
   DP_DIAG4[84] := B#16#0;
   DP_DIAG4[85] := B#16#0;
   DP_DIAG4[86] := B#16#0;
   DP_DIAG4[87] := B#16#0;
   DP_DIAG4[88] := B#16#0;
   DP_DIAG4[89] := B#16#0;
   DP_DIAG4[90] := B#16#0;
   DP_DIAG4[91] := B#16#0;
   DP_DIAG4[92] := B#16#0;
   DP_DIAG4[93] := B#16#0;
   DP_DIAG4[94] := B#16#0;
   DP_DIAG4[95] := B#16#0;
   DP_DIAG4[96] := B#16#0;
   DP_DIAG4[97] := B#16#0;
   DP_DIAG4[98] := B#16#0;
   DP_DIAG4[99] := B#16#0;
   DP_DIAG4[100] := B#16#0;
   DP_DIAG5[1] := B#16#0;
   DP_DIAG5[2] := B#16#0;
   DP_DIAG5[3] := B#16#0;
   DP_DIAG5[4] := B#16#0;
   DP_DIAG5[5] := B#16#0;
   DP_DIAG5[6] := B#16#0;
   DP_DIAG5[7] := B#16#0;
   DP_DIAG5[8] := B#16#0;
   DP_DIAG5[9] := B#16#0;
   DP_DIAG5[10] := B#16#0;
   DP_DIAG5[11] := B#16#0;
   DP_DIAG5[12] := B#16#0;
   DP_DIAG5[13] := B#16#0;
   DP_DIAG5[14] := B#16#0;
   DP_DIAG5[15] := B#16#0;
   DP_DIAG5[16] := B#16#0;
   DP_DIAG5[17] := B#16#0;
   DP_DIAG5[18] := B#16#0;
   DP_DIAG5[19] := B#16#0;
   DP_DIAG5[20] := B#16#0;
   DP_DIAG5[21] := B#16#0;
   DP_DIAG5[22] := B#16#0;
   DP_DIAG5[23] := B#16#0;
   DP_DIAG5[24] := B#16#0;
   DP_DIAG5[25] := B#16#0;
   DP_DIAG5[26] := B#16#0;
   DP_DIAG5[27] := B#16#0;
   DP_DIAG5[28] := B#16#0;
   DP_DIAG5[29] := B#16#0;
   DP_DIAG5[30] := B#16#0;
   DP_DIAG5[31] := B#16#0;
   DP_DIAG5[32] := B#16#0;
   DP_DIAG5[33] := B#16#0;
   DP_DIAG5[34] := B#16#0;
   DP_DIAG5[35] := B#16#0;
   DP_DIAG5[36] := B#16#0;
   DP_DIAG5[37] := B#16#0;
   DP_DIAG5[38] := B#16#0;
   DP_DIAG5[39] := B#16#0;
   DP_DIAG5[40] := B#16#0;
   DP_DIAG5[41] := B#16#0;
   DP_DIAG5[42] := B#16#0;
   DP_DIAG5[43] := B#16#0;
   DP_DIAG5[44] := B#16#0;
   DP_DIAG5[45] := B#16#0;
   DP_DIAG5[46] := B#16#0;
   DP_DIAG5[47] := B#16#0;
   DP_DIAG5[48] := B#16#0;
   DP_DIAG5[49] := B#16#0;
   DP_DIAG5[50] := B#16#0;
   DP_DIAG5[51] := B#16#0;
   DP_DIAG5[52] := B#16#0;
   DP_DIAG5[53] := B#16#0;
   DP_DIAG5[54] := B#16#0;
   DP_DIAG5[55] := B#16#0;
   DP_DIAG5[56] := B#16#0;
   DP_DIAG5[57] := B#16#0;
   DP_DIAG5[58] := B#16#0;
   DP_DIAG5[59] := B#16#0;
   DP_DIAG5[60] := B#16#0;
   DP_DIAG5[61] := B#16#0;
   DP_DIAG5[62] := B#16#0;
   DP_DIAG5[63] := B#16#0;
   DP_DIAG5[64] := B#16#0;
   DP_DIAG5[65] := B#16#0;
   DP_DIAG5[66] := B#16#0;
   DP_DIAG5[67] := B#16#0;
   DP_DIAG5[68] := B#16#0;
   DP_DIAG5[69] := B#16#0;
   DP_DIAG5[70] := B#16#0;
   DP_DIAG5[71] := B#16#0;
   DP_DIAG5[72] := B#16#0;
   DP_DIAG5[73] := B#16#0;
   DP_DIAG5[74] := B#16#0;
   DP_DIAG5[75] := B#16#0;
   DP_DIAG5[76] := B#16#0;
   DP_DIAG5[77] := B#16#0;
   DP_DIAG5[78] := B#16#0;
   DP_DIAG5[79] := B#16#0;
   DP_DIAG5[80] := B#16#0;
   DP_DIAG5[81] := B#16#0;
   DP_DIAG5[82] := B#16#0;
   DP_DIAG5[83] := B#16#0;
   DP_DIAG5[84] := B#16#0;
   DP_DIAG5[85] := B#16#0;
   DP_DIAG5[86] := B#16#0;
   DP_DIAG5[87] := B#16#0;
   DP_DIAG5[88] := B#16#0;
   DP_DIAG5[89] := B#16#0;
   DP_DIAG5[90] := B#16#0;
   DP_DIAG5[91] := B#16#0;
   DP_DIAG5[92] := B#16#0;
   DP_DIAG5[93] := B#16#0;
   DP_DIAG5[94] := B#16#0;
   DP_DIAG5[95] := B#16#0;
   DP_DIAG5[96] := B#16#0;
   DP_DIAG5[97] := B#16#0;
   DP_DIAG5[98] := B#16#0;
   DP_DIAG5[99] := B#16#0;
   DP_DIAG5[100] := B#16#0;
   DP_DIAG6[1] := B#16#0;
   DP_DIAG6[2] := B#16#0;
   DP_DIAG6[3] := B#16#0;
   DP_DIAG6[4] := B#16#0;
   DP_DIAG6[5] := B#16#0;
   DP_DIAG6[6] := B#16#0;
   DP_DIAG6[7] := B#16#0;
   DP_DIAG6[8] := B#16#0;
   DP_DIAG6[9] := B#16#0;
   DP_DIAG6[10] := B#16#0;
   DP_DIAG6[11] := B#16#0;
   DP_DIAG6[12] := B#16#0;
   DP_DIAG6[13] := B#16#0;
   DP_DIAG6[14] := B#16#0;
   DP_DIAG6[15] := B#16#0;
   DP_DIAG6[16] := B#16#0;
   DP_DIAG6[17] := B#16#0;
   DP_DIAG6[18] := B#16#0;
   DP_DIAG6[19] := B#16#0;
   DP_DIAG6[20] := B#16#0;
   DP_DIAG6[21] := B#16#0;
   DP_DIAG6[22] := B#16#0;
   DP_DIAG6[23] := B#16#0;
   DP_DIAG6[24] := B#16#0;
   DP_DIAG6[25] := B#16#0;
   DP_DIAG6[26] := B#16#0;
   DP_DIAG6[27] := B#16#0;
   DP_DIAG6[28] := B#16#0;
   DP_DIAG6[29] := B#16#0;
   DP_DIAG6[30] := B#16#0;
   DP_DIAG6[31] := B#16#0;
   DP_DIAG6[32] := B#16#0;
   DP_DIAG6[33] := B#16#0;
   DP_DIAG6[34] := B#16#0;
   DP_DIAG6[35] := B#16#0;
   DP_DIAG6[36] := B#16#0;
   DP_DIAG6[37] := B#16#0;
   DP_DIAG6[38] := B#16#0;
   DP_DIAG6[39] := B#16#0;
   DP_DIAG6[40] := B#16#0;
   DP_DIAG6[41] := B#16#0;
   DP_DIAG6[42] := B#16#0;
   DP_DIAG6[43] := B#16#0;
   DP_DIAG6[44] := B#16#0;
   DP_DIAG6[45] := B#16#0;
   DP_DIAG6[46] := B#16#0;
   DP_DIAG6[47] := B#16#0;
   DP_DIAG6[48] := B#16#0;
   DP_DIAG6[49] := B#16#0;
   DP_DIAG6[50] := B#16#0;
   DP_DIAG6[51] := B#16#0;
   DP_DIAG6[52] := B#16#0;
   DP_DIAG6[53] := B#16#0;
   DP_DIAG6[54] := B#16#0;
   DP_DIAG6[55] := B#16#0;
   DP_DIAG6[56] := B#16#0;
   DP_DIAG6[57] := B#16#0;
   DP_DIAG6[58] := B#16#0;
   DP_DIAG6[59] := B#16#0;
   DP_DIAG6[60] := B#16#0;
   DP_DIAG6[61] := B#16#0;
   DP_DIAG6[62] := B#16#0;
   DP_DIAG6[63] := B#16#0;
   DP_DIAG6[64] := B#16#0;
   DP_DIAG6[65] := B#16#0;
   DP_DIAG6[66] := B#16#0;
   DP_DIAG6[67] := B#16#0;
   DP_DIAG6[68] := B#16#0;
   DP_DIAG6[69] := B#16#0;
   DP_DIAG6[70] := B#16#0;
   DP_DIAG6[71] := B#16#0;
   DP_DIAG6[72] := B#16#0;
   DP_DIAG6[73] := B#16#0;
   DP_DIAG6[74] := B#16#0;
   DP_DIAG6[75] := B#16#0;
   DP_DIAG6[76] := B#16#0;
   DP_DIAG6[77] := B#16#0;
   DP_DIAG6[78] := B#16#0;
   DP_DIAG6[79] := B#16#0;
   DP_DIAG6[80] := B#16#0;
   DP_DIAG6[81] := B#16#0;
   DP_DIAG6[82] := B#16#0;
   DP_DIAG6[83] := B#16#0;
   DP_DIAG6[84] := B#16#0;
   DP_DIAG6[85] := B#16#0;
   DP_DIAG6[86] := B#16#0;
   DP_DIAG6[87] := B#16#0;
   DP_DIAG6[88] := B#16#0;
   DP_DIAG6[89] := B#16#0;
   DP_DIAG6[90] := B#16#0;
   DP_DIAG6[91] := B#16#0;
   DP_DIAG6[92] := B#16#0;
   DP_DIAG6[93] := B#16#0;
   DP_DIAG6[94] := B#16#0;
   DP_DIAG6[95] := B#16#0;
   DP_DIAG6[96] := B#16#0;
   DP_DIAG6[97] := B#16#0;
   DP_DIAG6[98] := B#16#0;
   DP_DIAG6[99] := B#16#0;
   DP_DIAG6[100] := B#16#0;
   DP_DIAG7[1] := B#16#0;
   DP_DIAG7[2] := B#16#0;
   DP_DIAG7[3] := B#16#0;
   DP_DIAG7[4] := B#16#0;
   DP_DIAG7[5] := B#16#0;
   DP_DIAG7[6] := B#16#0;
   DP_DIAG7[7] := B#16#0;
   DP_DIAG7[8] := B#16#0;
   DP_DIAG7[9] := B#16#0;
   DP_DIAG7[10] := B#16#0;
   DP_DIAG7[11] := B#16#0;
   DP_DIAG7[12] := B#16#0;
   DP_DIAG7[13] := B#16#0;
   DP_DIAG7[14] := B#16#0;
   DP_DIAG7[15] := B#16#0;
   DP_DIAG7[16] := B#16#0;
   DP_DIAG7[17] := B#16#0;
   DP_DIAG7[18] := B#16#0;
   DP_DIAG7[19] := B#16#0;
   DP_DIAG7[20] := B#16#0;
   DP_DIAG7[21] := B#16#0;
   DP_DIAG7[22] := B#16#0;
   DP_DIAG7[23] := B#16#0;
   DP_DIAG7[24] := B#16#0;
   DP_DIAG7[25] := B#16#0;
   DP_DIAG7[26] := B#16#0;
   DP_DIAG7[27] := B#16#0;
   DP_DIAG7[28] := B#16#0;
   DP_DIAG7[29] := B#16#0;
   DP_DIAG7[30] := B#16#0;
   DP_DIAG7[31] := B#16#0;
   DP_DIAG7[32] := B#16#0;
   DP_DIAG7[33] := B#16#0;
   DP_DIAG7[34] := B#16#0;
   DP_DIAG7[35] := B#16#0;
   DP_DIAG7[36] := B#16#0;
   DP_DIAG7[37] := B#16#0;
   DP_DIAG7[38] := B#16#0;
   DP_DIAG7[39] := B#16#0;
   DP_DIAG7[40] := B#16#0;
   DP_DIAG7[41] := B#16#0;
   DP_DIAG7[42] := B#16#0;
   DP_DIAG7[43] := B#16#0;
   DP_DIAG7[44] := B#16#0;
   DP_DIAG7[45] := B#16#0;
   DP_DIAG7[46] := B#16#0;
   DP_DIAG7[47] := B#16#0;
   DP_DIAG7[48] := B#16#0;
   DP_DIAG7[49] := B#16#0;
   DP_DIAG7[50] := B#16#0;
   DP_DIAG7[51] := B#16#0;
   DP_DIAG7[52] := B#16#0;
   DP_DIAG7[53] := B#16#0;
   DP_DIAG7[54] := B#16#0;
   DP_DIAG7[55] := B#16#0;
   DP_DIAG7[56] := B#16#0;
   DP_DIAG7[57] := B#16#0;
   DP_DIAG7[58] := B#16#0;
   DP_DIAG7[59] := B#16#0;
   DP_DIAG7[60] := B#16#0;
   DP_DIAG7[61] := B#16#0;
   DP_DIAG7[62] := B#16#0;
   DP_DIAG7[63] := B#16#0;
   DP_DIAG7[64] := B#16#0;
   DP_DIAG7[65] := B#16#0;
   DP_DIAG7[66] := B#16#0;
   DP_DIAG7[67] := B#16#0;
   DP_DIAG7[68] := B#16#0;
   DP_DIAG7[69] := B#16#0;
   DP_DIAG7[70] := B#16#0;
   DP_DIAG7[71] := B#16#0;
   DP_DIAG7[72] := B#16#0;
   DP_DIAG7[73] := B#16#0;
   DP_DIAG7[74] := B#16#0;
   DP_DIAG7[75] := B#16#0;
   DP_DIAG7[76] := B#16#0;
   DP_DIAG7[77] := B#16#0;
   DP_DIAG7[78] := B#16#0;
   DP_DIAG7[79] := B#16#0;
   DP_DIAG7[80] := B#16#0;
   DP_DIAG7[81] := B#16#0;
   DP_DIAG7[82] := B#16#0;
   DP_DIAG7[83] := B#16#0;
   DP_DIAG7[84] := B#16#0;
   DP_DIAG7[85] := B#16#0;
   DP_DIAG7[86] := B#16#0;
   DP_DIAG7[87] := B#16#0;
   DP_DIAG7[88] := B#16#0;
   DP_DIAG7[89] := B#16#0;
   DP_DIAG7[90] := B#16#0;
   DP_DIAG7[91] := B#16#0;
   DP_DIAG7[92] := B#16#0;
   DP_DIAG7[93] := B#16#0;
   DP_DIAG7[94] := B#16#0;
   DP_DIAG7[95] := B#16#0;
   DP_DIAG7[96] := B#16#0;
   DP_DIAG7[97] := B#16#0;
   DP_DIAG7[98] := B#16#0;
   DP_DIAG7[99] := B#16#0;
   DP_DIAG7[100] := B#16#0;
   DP_DIAG8[1] := B#16#0;
   DP_DIAG8[2] := B#16#0;
   DP_DIAG8[3] := B#16#0;
   DP_DIAG8[4] := B#16#0;
   DP_DIAG8[5] := B#16#0;
   DP_DIAG8[6] := B#16#0;
   DP_DIAG8[7] := B#16#0;
   DP_DIAG8[8] := B#16#0;
   DP_DIAG8[9] := B#16#0;
   DP_DIAG8[10] := B#16#0;
   DP_DIAG8[11] := B#16#0;
   DP_DIAG8[12] := B#16#0;
   DP_DIAG8[13] := B#16#0;
   DP_DIAG8[14] := B#16#0;
   DP_DIAG8[15] := B#16#0;
   DP_DIAG8[16] := B#16#0;
   DP_DIAG8[17] := B#16#0;
   DP_DIAG8[18] := B#16#0;
   DP_DIAG8[19] := B#16#0;
   DP_DIAG8[20] := B#16#0;
   DP_DIAG8[21] := B#16#0;
   DP_DIAG8[22] := B#16#0;
   DP_DIAG8[23] := B#16#0;
   DP_DIAG8[24] := B#16#0;
   DP_DIAG8[25] := B#16#0;
   DP_DIAG8[26] := B#16#0;
   DP_DIAG8[27] := B#16#0;
   DP_DIAG8[28] := B#16#0;
   DP_DIAG8[29] := B#16#0;
   DP_DIAG8[30] := B#16#0;
   DP_DIAG8[31] := B#16#0;
   DP_DIAG8[32] := B#16#0;
   DP_DIAG8[33] := B#16#0;
   DP_DIAG8[34] := B#16#0;
   DP_DIAG8[35] := B#16#0;
   DP_DIAG8[36] := B#16#0;
   DP_DIAG8[37] := B#16#0;
   DP_DIAG8[38] := B#16#0;
   DP_DIAG8[39] := B#16#0;
   DP_DIAG8[40] := B#16#0;
   DP_DIAG8[41] := B#16#0;
   DP_DIAG8[42] := B#16#0;
   DP_DIAG8[43] := B#16#0;
   DP_DIAG8[44] := B#16#0;
   DP_DIAG8[45] := B#16#0;
   DP_DIAG8[46] := B#16#0;
   DP_DIAG8[47] := B#16#0;
   DP_DIAG8[48] := B#16#0;
   DP_DIAG8[49] := B#16#0;
   DP_DIAG8[50] := B#16#0;
   DP_DIAG8[51] := B#16#0;
   DP_DIAG8[52] := B#16#0;
   DP_DIAG8[53] := B#16#0;
   DP_DIAG8[54] := B#16#0;
   DP_DIAG8[55] := B#16#0;
   DP_DIAG8[56] := B#16#0;
   DP_DIAG8[57] := B#16#0;
   DP_DIAG8[58] := B#16#0;
   DP_DIAG8[59] := B#16#0;
   DP_DIAG8[60] := B#16#0;
   DP_DIAG8[61] := B#16#0;
   DP_DIAG8[62] := B#16#0;
   DP_DIAG8[63] := B#16#0;
   DP_DIAG8[64] := B#16#0;
   DP_DIAG8[65] := B#16#0;
   DP_DIAG8[66] := B#16#0;
   DP_DIAG8[67] := B#16#0;
   DP_DIAG8[68] := B#16#0;
   DP_DIAG8[69] := B#16#0;
   DP_DIAG8[70] := B#16#0;
   DP_DIAG8[71] := B#16#0;
   DP_DIAG8[72] := B#16#0;
   DP_DIAG8[73] := B#16#0;
   DP_DIAG8[74] := B#16#0;
   DP_DIAG8[75] := B#16#0;
   DP_DIAG8[76] := B#16#0;
   DP_DIAG8[77] := B#16#0;
   DP_DIAG8[78] := B#16#0;
   DP_DIAG8[79] := B#16#0;
   DP_DIAG8[80] := B#16#0;
   DP_DIAG8[81] := B#16#0;
   DP_DIAG8[82] := B#16#0;
   DP_DIAG8[83] := B#16#0;
   DP_DIAG8[84] := B#16#0;
   DP_DIAG8[85] := B#16#0;
   DP_DIAG8[86] := B#16#0;
   DP_DIAG8[87] := B#16#0;
   DP_DIAG8[88] := B#16#0;
   DP_DIAG8[89] := B#16#0;
   DP_DIAG8[90] := B#16#0;
   DP_DIAG8[91] := B#16#0;
   DP_DIAG8[92] := B#16#0;
   DP_DIAG8[93] := B#16#0;
   DP_DIAG8[94] := B#16#0;
   DP_DIAG8[95] := B#16#0;
   DP_DIAG8[96] := B#16#0;
   DP_DIAG8[97] := B#16#0;
   DP_DIAG8[98] := B#16#0;
   DP_DIAG8[99] := B#16#0;
   DP_DIAG8[100] := B#16#0;
   DP_DIAG9[1] := B#16#0;
   DP_DIAG9[2] := B#16#0;
   DP_DIAG9[3] := B#16#0;
   DP_DIAG9[4] := B#16#0;
   DP_DIAG9[5] := B#16#0;
   DP_DIAG9[6] := B#16#0;
   DP_DIAG9[7] := B#16#0;
   DP_DIAG9[8] := B#16#0;
   DP_DIAG9[9] := B#16#0;
   DP_DIAG9[10] := B#16#0;
   DP_DIAG9[11] := B#16#0;
   DP_DIAG9[12] := B#16#0;
   DP_DIAG9[13] := B#16#0;
   DP_DIAG9[14] := B#16#0;
   DP_DIAG9[15] := B#16#0;
   DP_DIAG9[16] := B#16#0;
   DP_DIAG9[17] := B#16#0;
   DP_DIAG9[18] := B#16#0;
   DP_DIAG9[19] := B#16#0;
   DP_DIAG9[20] := B#16#0;
   DP_DIAG9[21] := B#16#0;
   DP_DIAG9[22] := B#16#0;
   DP_DIAG9[23] := B#16#0;
   DP_DIAG9[24] := B#16#0;
   DP_DIAG9[25] := B#16#0;
   DP_DIAG9[26] := B#16#0;
   DP_DIAG9[27] := B#16#0;
   DP_DIAG9[28] := B#16#0;
   DP_DIAG9[29] := B#16#0;
   DP_DIAG9[30] := B#16#0;
   DP_DIAG9[31] := B#16#0;
   DP_DIAG9[32] := B#16#0;
   DP_DIAG9[33] := B#16#0;
   DP_DIAG9[34] := B#16#0;
   DP_DIAG9[35] := B#16#0;
   DP_DIAG9[36] := B#16#0;
   DP_DIAG9[37] := B#16#0;
   DP_DIAG9[38] := B#16#0;
   DP_DIAG9[39] := B#16#0;
   DP_DIAG9[40] := B#16#0;
   DP_DIAG9[41] := B#16#0;
   DP_DIAG9[42] := B#16#0;
   DP_DIAG9[43] := B#16#0;
   DP_DIAG9[44] := B#16#0;
   DP_DIAG9[45] := B#16#0;
   DP_DIAG9[46] := B#16#0;
   DP_DIAG9[47] := B#16#0;
   DP_DIAG9[48] := B#16#0;
   DP_DIAG9[49] := B#16#0;
   DP_DIAG9[50] := B#16#0;
   DP_DIAG9[51] := B#16#0;
   DP_DIAG9[52] := B#16#0;
   DP_DIAG9[53] := B#16#0;
   DP_DIAG9[54] := B#16#0;
   DP_DIAG9[55] := B#16#0;
   DP_DIAG9[56] := B#16#0;
   DP_DIAG9[57] := B#16#0;
   DP_DIAG9[58] := B#16#0;
   DP_DIAG9[59] := B#16#0;
   DP_DIAG9[60] := B#16#0;
   DP_DIAG9[61] := B#16#0;
   DP_DIAG9[62] := B#16#0;
   DP_DIAG9[63] := B#16#0;
   DP_DIAG9[64] := B#16#0;
   DP_DIAG9[65] := B#16#0;
   DP_DIAG9[66] := B#16#0;
   DP_DIAG9[67] := B#16#0;
   DP_DIAG9[68] := B#16#0;
   DP_DIAG9[69] := B#16#0;
   DP_DIAG9[70] := B#16#0;
   DP_DIAG9[71] := B#16#0;
   DP_DIAG9[72] := B#16#0;
   DP_DIAG9[73] := B#16#0;
   DP_DIAG9[74] := B#16#0;
   DP_DIAG9[75] := B#16#0;
   DP_DIAG9[76] := B#16#0;
   DP_DIAG9[77] := B#16#0;
   DP_DIAG9[78] := B#16#0;
   DP_DIAG9[79] := B#16#0;
   DP_DIAG9[80] := B#16#0;
   DP_DIAG9[81] := B#16#0;
   DP_DIAG9[82] := B#16#0;
   DP_DIAG9[83] := B#16#0;
   DP_DIAG9[84] := B#16#0;
   DP_DIAG9[85] := B#16#0;
   DP_DIAG9[86] := B#16#0;
   DP_DIAG9[87] := B#16#0;
   DP_DIAG9[88] := B#16#0;
   DP_DIAG9[89] := B#16#0;
   DP_DIAG9[90] := B#16#0;
   DP_DIAG9[91] := B#16#0;
   DP_DIAG9[92] := B#16#0;
   DP_DIAG9[93] := B#16#0;
   DP_DIAG9[94] := B#16#0;
   DP_DIAG9[95] := B#16#0;
   DP_DIAG9[96] := B#16#0;
   DP_DIAG9[97] := B#16#0;
   DP_DIAG9[98] := B#16#0;
   DP_DIAG9[99] := B#16#0;
   DP_DIAG9[100] := B#16#0;
   DP_DIAG10[1] := B#16#0;
   DP_DIAG10[2] := B#16#0;
   DP_DIAG10[3] := B#16#0;
   DP_DIAG10[4] := B#16#0;
   DP_DIAG10[5] := B#16#0;
   DP_DIAG10[6] := B#16#0;
   DP_DIAG10[7] := B#16#0;
   DP_DIAG10[8] := B#16#0;
   DP_DIAG10[9] := B#16#0;
   DP_DIAG10[10] := B#16#0;
   DP_DIAG10[11] := B#16#0;
   DP_DIAG10[12] := B#16#0;
   DP_DIAG10[13] := B#16#0;
   DP_DIAG10[14] := B#16#0;
   DP_DIAG10[15] := B#16#0;
   DP_DIAG10[16] := B#16#0;
   DP_DIAG10[17] := B#16#0;
   DP_DIAG10[18] := B#16#0;
   DP_DIAG10[19] := B#16#0;
   DP_DIAG10[20] := B#16#0;
   DP_DIAG10[21] := B#16#0;
   DP_DIAG10[22] := B#16#0;
   DP_DIAG10[23] := B#16#0;
   DP_DIAG10[24] := B#16#0;
   DP_DIAG10[25] := B#16#0;
   DP_DIAG10[26] := B#16#0;
   DP_DIAG10[27] := B#16#0;
   DP_DIAG10[28] := B#16#0;
   DP_DIAG10[29] := B#16#0;
   DP_DIAG10[30] := B#16#0;
   DP_DIAG10[31] := B#16#0;
   DP_DIAG10[32] := B#16#0;
   DP_DIAG10[33] := B#16#0;
   DP_DIAG10[34] := B#16#0;
   DP_DIAG10[35] := B#16#0;
   DP_DIAG10[36] := B#16#0;
   DP_DIAG10[37] := B#16#0;
   DP_DIAG10[38] := B#16#0;
   DP_DIAG10[39] := B#16#0;
   DP_DIAG10[40] := B#16#0;
   DP_DIAG10[41] := B#16#0;
   DP_DIAG10[42] := B#16#0;
   DP_DIAG10[43] := B#16#0;
   DP_DIAG10[44] := B#16#0;
   DP_DIAG10[45] := B#16#0;
   DP_DIAG10[46] := B#16#0;
   DP_DIAG10[47] := B#16#0;
   DP_DIAG10[48] := B#16#0;
   DP_DIAG10[49] := B#16#0;
   DP_DIAG10[50] := B#16#0;
   DP_DIAG10[51] := B#16#0;
   DP_DIAG10[52] := B#16#0;
   DP_DIAG10[53] := B#16#0;
   DP_DIAG10[54] := B#16#0;
   DP_DIAG10[55] := B#16#0;
   DP_DIAG10[56] := B#16#0;
   DP_DIAG10[57] := B#16#0;
   DP_DIAG10[58] := B#16#0;
   DP_DIAG10[59] := B#16#0;
   DP_DIAG10[60] := B#16#0;
   DP_DIAG10[61] := B#16#0;
   DP_DIAG10[62] := B#16#0;
   DP_DIAG10[63] := B#16#0;
   DP_DIAG10[64] := B#16#0;
   DP_DIAG10[65] := B#16#0;
   DP_DIAG10[66] := B#16#0;
   DP_DIAG10[67] := B#16#0;
   DP_DIAG10[68] := B#16#0;
   DP_DIAG10[69] := B#16#0;
   DP_DIAG10[70] := B#16#0;
   DP_DIAG10[71] := B#16#0;
   DP_DIAG10[72] := B#16#0;
   DP_DIAG10[73] := B#16#0;
   DP_DIAG10[74] := B#16#0;
   DP_DIAG10[75] := B#16#0;
   DP_DIAG10[76] := B#16#0;
   DP_DIAG10[77] := B#16#0;
   DP_DIAG10[78] := B#16#0;
   DP_DIAG10[79] := B#16#0;
   DP_DIAG10[80] := B#16#0;
   DP_DIAG10[81] := B#16#0;
   DP_DIAG10[82] := B#16#0;
   DP_DIAG10[83] := B#16#0;
   DP_DIAG10[84] := B#16#0;
   DP_DIAG10[85] := B#16#0;
   DP_DIAG10[86] := B#16#0;
   DP_DIAG10[87] := B#16#0;
   DP_DIAG10[88] := B#16#0;
   DP_DIAG10[89] := B#16#0;
   DP_DIAG10[90] := B#16#0;
   DP_DIAG10[91] := B#16#0;
   DP_DIAG10[92] := B#16#0;
   DP_DIAG10[93] := B#16#0;
   DP_DIAG10[94] := B#16#0;
   DP_DIAG10[95] := B#16#0;
   DP_DIAG10[96] := B#16#0;
   DP_DIAG10[97] := B#16#0;
   DP_DIAG10[98] := B#16#0;
   DP_DIAG10[99] := B#16#0;
   DP_DIAG10[100] := B#16#0;
END_DATA_BLOCK

FUNCTION_BLOCK FB 402
TITLE =Operation Mode Select Program
AUTHOR : HMC
FAMILY : Mode
NAME : Mode
VERSION : 1.0


VAR_INPUT
  SSD_Manual : BOOL ;
  SSD_Auto : BOOL ;
  PB_Ready : BOOL ;
  PB_Auto_Run : BOOL ;
  PB_Remote_Ready : BOOL ;
  PB_Remote_Auto_Run : BOOL ;
  PB_Lamp_CHK : BOOL ;
  M_Air_Error : BOOL ;
  M_Water_Error : BOOL ;
  M_Total_Error : BOOL ;
  M_EStop : BOOL ;
  EXT_Ready : BOOL ;
  EXT_Auto : BOOL ;
  T_SemiAuto : TIME ;
  M_FLICK : BOOL ;
END_VAR
VAR_OUTPUT
  M_Ready_On : BOOL ;
  M_Auto_Mode : BOOL ;
  M_SemiAuto_Mode : BOOL ;
  M_Manual_Mode : BOOL ;
  M_Auto_Run : BOOL ;
  LP_Ready_On : BOOL ;
  LP_Auto_Run : BOOL ;
END_VAR
VAR
  AUTO_MODE_DELAY : SFB 4;
  SEMI_AUTO_DELAY : SFB 4;
  MANUAL_DELAY : SFB 4;
END_VAR
BEGIN
NETWORK
TITLE =Auto Mode Select Program
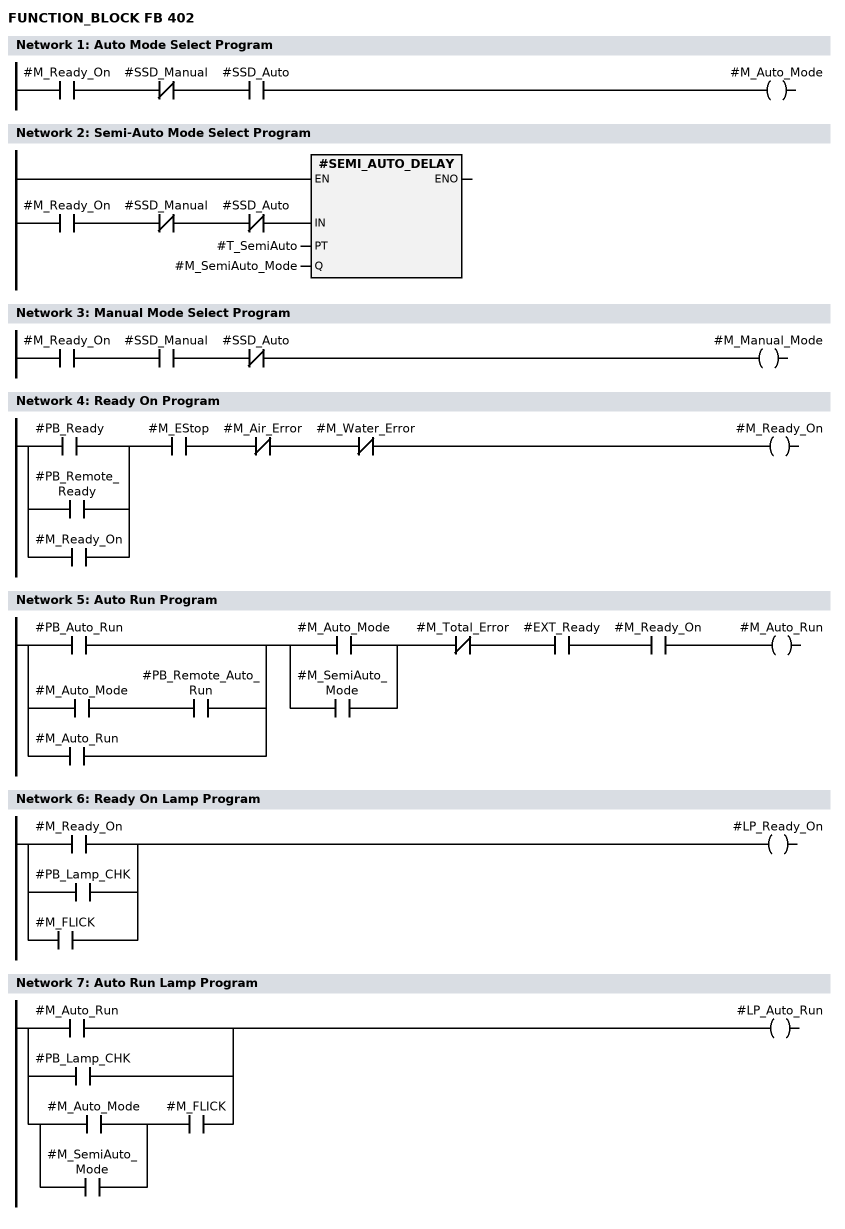

      A     #M_Ready_On;
      AN    #SSD_Manual;
      A     #SSD_Auto;
      =     #M_Auto_Mode;
NETWORK
TITLE =Semi-Auto Mode Select Program

      A     #M_Ready_On;
      AN    #SSD_Manual;
      AN    #SSD_Auto;
      =     L      0.0;
      BLD   103;
      CALL #SEMI_AUTO_DELAY (
           IN                       := L      0.0,
           PT                       := #T_SemiAuto,
           Q                        := #M_SemiAuto_Mode);

      NOP   0;
NETWORK
TITLE =Manual Mode Select Program

      A     #M_Ready_On;
      A     #SSD_Manual;
      AN    #SSD_Auto;
      =     #M_Manual_Mode;
NETWORK
TITLE =Ready On Program

      A(    ;
      O     #PB_Ready;
      O     #PB_Remote_Ready;
      O     #M_Ready_On;
      )     ;
      A     #M_EStop;
      AN    #M_Air_Error;
      AN    #M_Water_Error;
      =     #M_Ready_On;
NETWORK
TITLE =Auto Run Program

      A(    ;
      O     #PB_Auto_Run;
      O     ;
      A     #M_Auto_Mode;
      A     #PB_Remote_Auto_Run;
      O     #M_Auto_Run;
      )     ;
      A(    ;
      O     #M_Auto_Mode;
      O     #M_SemiAuto_Mode;
      )     ;
      AN    #M_Total_Error;
      A     #EXT_Ready;
      A     #M_Ready_On;
      =     #M_Auto_Run;
NETWORK
TITLE =Ready On Lamp Program

      O     #M_Ready_On;
      O     #PB_Lamp_CHK;
      O     #M_FLICK;
      =     #LP_Ready_On;
NETWORK
TITLE =Auto Run Lamp Program

      O     #M_Auto_Run;
      O     #PB_Lamp_CHK;
      O     ;
      A(    ;
      O     #M_Auto_Mode;
      O     #M_SemiAuto_Mode;
      )     ;
      A     #M_FLICK;
      =     #LP_Auto_Run;
END_FUNCTION_BLOCK

FUNCTION_BLOCK FB 424
TITLE =Sensor Error,Lamp Variables Program
AUTHOR : HMC
FAMILY : Common
NAME : Common
VERSION : 1.0


VAR_INPUT
  Enable_Aux : BOOL ;
  Adv_Amount : INT ;
  Ret_Amount : INT ;
  LS_Adv1 : BOOL ;
  LS_Ret1 : BOOL ;
  LS_Adv2 : BOOL ;
  LS_Ret2 : BOOL ;
  LS_Adv3 : BOOL ;
  LS_Ret3 : BOOL ;
  LS_Adv4 : BOOL ;
  LS_Ret4 : BOOL ;
  SOL_Adv : BOOL ;
  SOL_Ret : BOOL ;
  M_Ready : BOOL ;
  T_CHK1 : TIME ;
  T_CHK2 : TIME ;
  PB_Lamp_CHK : BOOL ;
  PB_Error_Rst : BOOL ;
  M_FLICK : BOOL ;
END_VAR
VAR_OUTPUT
  M_Adv_Err : BOOL ;
  M_Ret_Err : BOOL ;
  LP_Adv : BOOL ;
  LP_Ret : BOOL ;
  Visu_Adv : WORD ;
  Visu_Ret : WORD ;
END_VAR
VAR
  Error_T1 : SFB 4;
  Error_T2 : SFB 4;
  CHK_Aux1 : BOOL ;
  CHK_Aux2 : BOOL ;
  Error_T1_DN : BOOL ;
  Error_T2_DN : BOOL ;
  Adv_Memo : BOOL ;
  Visu_Adv_Arr : ARRAY  [0 .. 15 ] OF BOOL ;
  Visu_Ret_Arr : ARRAY  [0 .. 15 ] OF BOOL ;
  BLK_Move_Ret : INT ;
  Enable : BOOL ;
  Adv_End : BOOL ;
  Ret_End : BOOL ;
END_VAR
BEGIN
NETWORK
TITLE =
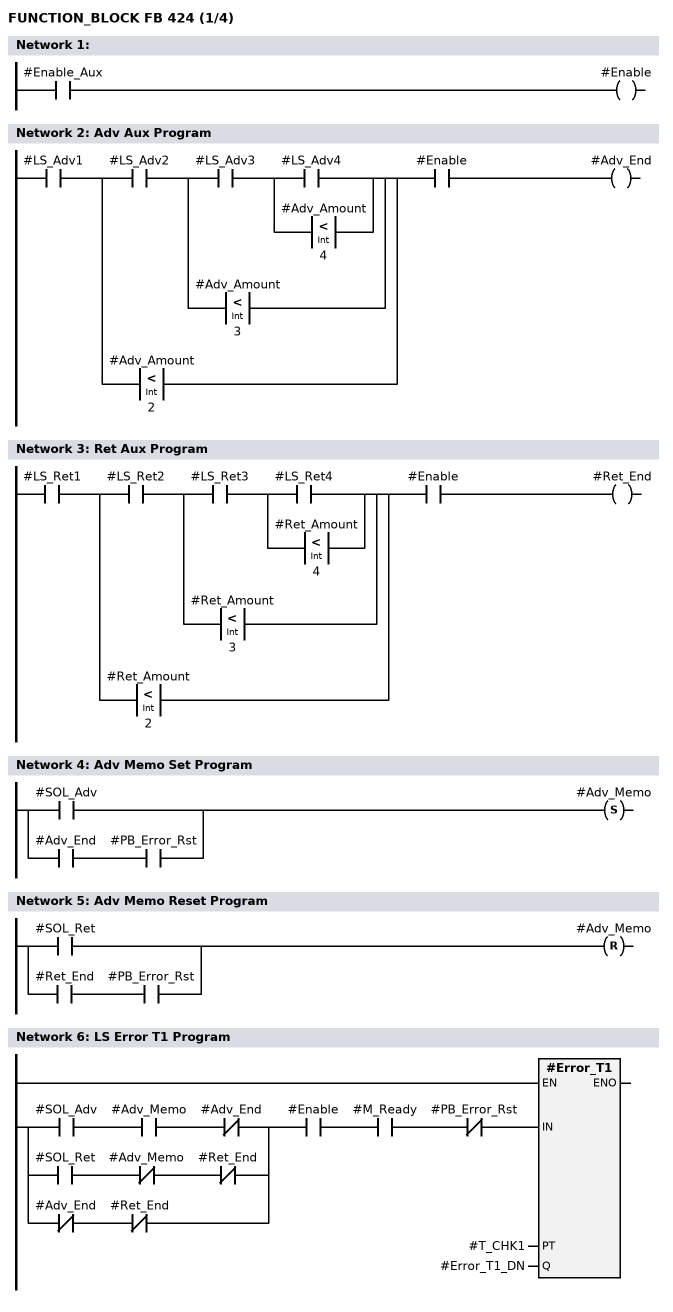

      A     #Enable_Aux;
      =     #Enable;
NETWORK
TITLE =Adv Aux Program

      A     #LS_Adv1;
      A(    ;
      A     #LS_Adv2;
      A(    ;
      A     #LS_Adv3;
      A(    ;
      O     #LS_Adv4;
      O(    ;
      L     #Adv_Amount;
      L     4;
      <I    ;
      )     ;
      )     ;
      O(    ;
      L     #Adv_Amount;
      L     3;
      <I    ;
      )     ;
      )     ;
      O(    ;
      L     #Adv_Amount;
      L     2;
      <I    ;
      )     ;
      )     ;
      A     #Enable;
      =     #Adv_End;
NETWORK
TITLE =Ret Aux Program

      A     #LS_Ret1;
      A(    ;
      A     #LS_Ret2;
      A(    ;
      A     #LS_Ret3;
      A(    ;
      O     #LS_Ret4;
      O(    ;
      L     #Ret_Amount;
      L     4;
      <I    ;
      )     ;
      )     ;
      O(    ;
      L     #Ret_Amount;
      L     3;
      <I    ;
      )     ;
      )     ;
      O(    ;
      L     #Ret_Amount;
      L     2;
      <I    ;
      )     ;
      )     ;
      A     #Enable;
      =     #Ret_End;
NETWORK
TITLE =Adv Memo Set Program

      O     #SOL_Adv;
      O     ;
      A     #Adv_End;
      A     #PB_Error_Rst;
      S     #Adv_Memo;
NETWORK
TITLE =Adv Memo Reset Program

      O     #SOL_Ret;
      O     ;
      A     #Ret_End;
      A     #PB_Error_Rst;
      R     #Adv_Memo;
NETWORK
TITLE =LS Error T1 Program

      A(    ;
      A     #SOL_Adv;
      A     #Adv_Memo;
      AN    #Adv_End;
      O     ;
      A     #SOL_Ret;
      AN    #Adv_Memo;
      AN    #Ret_End;
      O     ;
      AN    #Adv_End;
      AN    #Ret_End;
      )     ;
      A     #Enable;
      A     #M_Ready;
      AN    #PB_Error_Rst;
      =     L      0.0;
      BLD   103;
      CALL #Error_T1 (
           IN                       := L      0.0,
           PT                       := #T_CHK1,
           Q                        := #Error_T1_DN);

      NOP   0;
NETWORK
TITLE =Check Aux1 Program
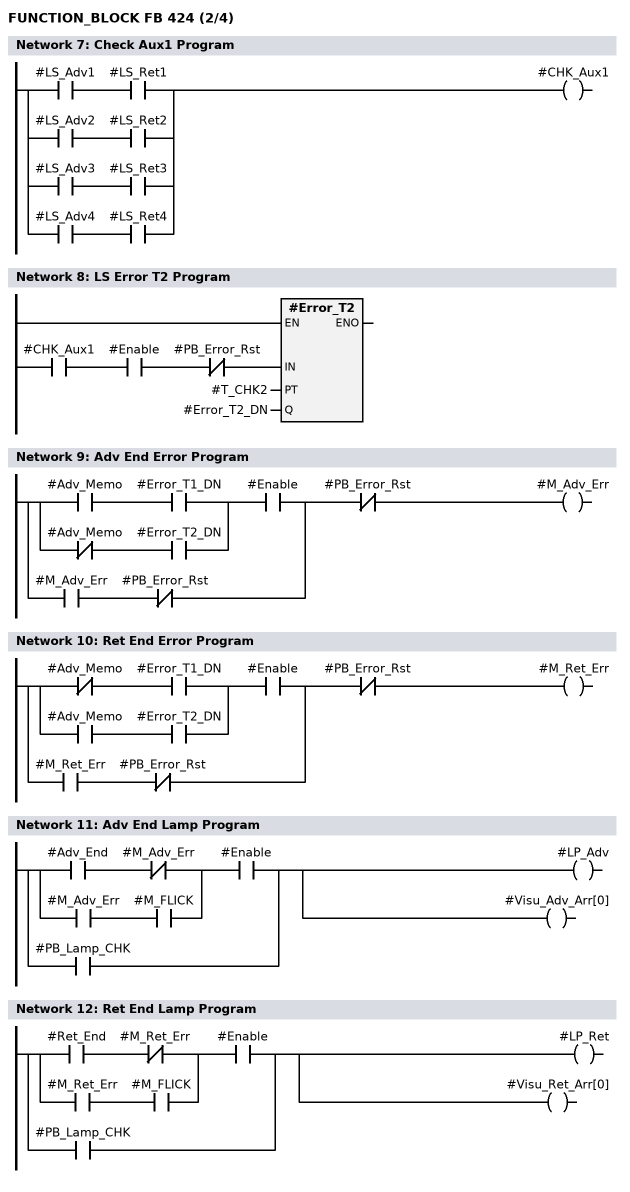

      A     #LS_Adv1;
      A     #LS_Ret1;
      O     ;
      A     #LS_Adv2;
      A     #LS_Ret2;
      O     ;
      A     #LS_Adv3;
      A     #LS_Ret3;
      O     ;
      A     #LS_Adv4;
      A     #LS_Ret4;
      =     #CHK_Aux1;
NETWORK
TITLE =LS Error T2 Program

      A     #CHK_Aux1;
      A     #Enable;
      AN    #PB_Error_Rst;
      =     L      0.0;
      BLD   103;
      CALL #Error_T2 (
           IN                       := L      0.0,
           PT                       := #T_CHK2,
           Q                        := #Error_T2_DN);

      NOP   0;
NETWORK
TITLE =Adv End Error Program

      A(    ;
      A(    ;
      A     #Adv_Memo;
      A     #Error_T1_DN;
      O     ;
      AN    #Adv_Memo;
      A     #Error_T2_DN;
      )     ;
      A     #Enable;
      O     ;
      A     #M_Adv_Err;
      AN    #PB_Error_Rst;
      )     ;
      AN    #PB_Error_Rst;
      =     #M_Adv_Err;
NETWORK
TITLE =Ret End Error Program

      A(    ;
      A(    ;
      AN    #Adv_Memo;
      A     #Error_T1_DN;
      O     ;
      A     #Adv_Memo;
      A     #Error_T2_DN;
      )     ;
      A     #Enable;
      O     ;
      A     #M_Ret_Err;
      AN    #PB_Error_Rst;
      )     ;
      AN    #PB_Error_Rst;
      =     #M_Ret_Err;
NETWORK
TITLE =Adv End Lamp Program

      A(    ;
      A     #Adv_End;
      AN    #M_Adv_Err;
      O     ;
      A     #M_Adv_Err;
      A     #M_FLICK;
      )     ;
      A     #Enable;
      O     #PB_Lamp_CHK;
      =     #LP_Adv;
      =     #Visu_Adv_Arr[0];
NETWORK
TITLE =Ret End Lamp Program

      A(    ;
      A     #Ret_End;
      AN    #M_Ret_Err;
      O     ;
      A     #M_Ret_Err;
      A     #M_FLICK;
      )     ;
      A     #Enable;
      O     #PB_Lamp_CHK;
      =     #LP_Ret;
      =     #Visu_Ret_Arr[0];
NETWORK
TITLE =Adv LS_1 Lamp Program
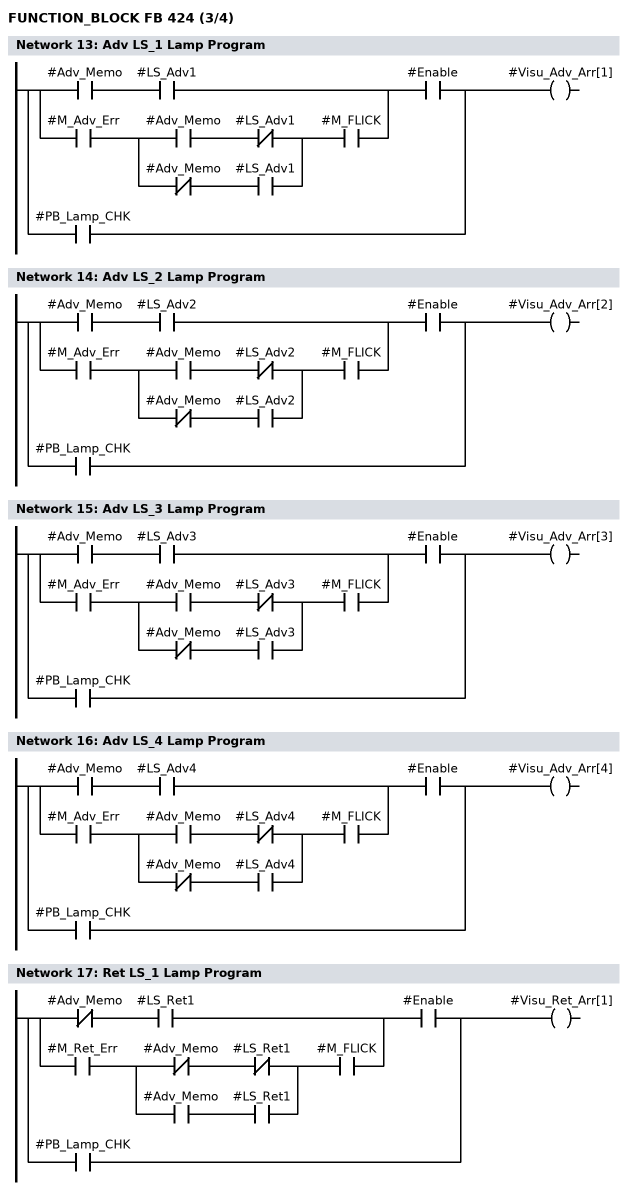

      A(    ;
      A     #Adv_Memo;
      A     #LS_Adv1;
      O     ;
      A     #M_Adv_Err;
      A(    ;
      A     #Adv_Memo;
      AN    #LS_Adv1;
      O     ;
      AN    #Adv_Memo;
      A     #LS_Adv1;
      )     ;
      A     #M_FLICK;
      )     ;
      A     #Enable;
      O     #PB_Lamp_CHK;
      =     #Visu_Adv_Arr[1];
NETWORK
TITLE =Adv LS_2 Lamp Program
//
//
      A(    ;
      A     #Adv_Memo;
      A     #LS_Adv2;
      O     ;
      A     #M_Adv_Err;
      A(    ;
      A     #Adv_Memo;
      AN    #LS_Adv2;
      O     ;
      AN    #Adv_Memo;
      A     #LS_Adv2;
      )     ;
      A     #M_FLICK;
      )     ;
      A     #Enable;
      O     #PB_Lamp_CHK;
      =     #Visu_Adv_Arr[2];
NETWORK
TITLE =Adv LS_3 Lamp Program
//
//
      A(    ;
      A     #Adv_Memo;
      A     #LS_Adv3;
      O     ;
      A     #M_Adv_Err;
      A(    ;
      A     #Adv_Memo;
      AN    #LS_Adv3;
      O     ;
      AN    #Adv_Memo;
      A     #LS_Adv3;
      )     ;
      A     #M_FLICK;
      )     ;
      A     #Enable;
      O     #PB_Lamp_CHK;
      =     #Visu_Adv_Arr[3];
NETWORK
TITLE =Adv LS_4 Lamp Program
//
//
      A(    ;
      A     #Adv_Memo;
      A     #LS_Adv4;
      O     ;
      A     #M_Adv_Err;
      A(    ;
      A     #Adv_Memo;
      AN    #LS_Adv4;
      O     ;
      AN    #Adv_Memo;
      A     #LS_Adv4;
      )     ;
      A     #M_FLICK;
      )     ;
      A     #Enable;
      O     #PB_Lamp_CHK;
      =     #Visu_Adv_Arr[4];
NETWORK
TITLE =Ret LS_1 Lamp Program
//
//
      A(    ;
      AN    #Adv_Memo;
      A     #LS_Ret1;
      O     ;
      A     #M_Ret_Err;
      A(    ;
      AN    #Adv_Memo;
      AN    #LS_Ret1;
      O     ;
      A     #Adv_Memo;
      A     #LS_Ret1;
      )     ;
      A     #M_FLICK;
      )     ;
      A     #Enable;
      O     #PB_Lamp_CHK;
      =     #Visu_Ret_Arr[1];
NETWORK
TITLE =Ret LS_2 Lamp Program
//
//
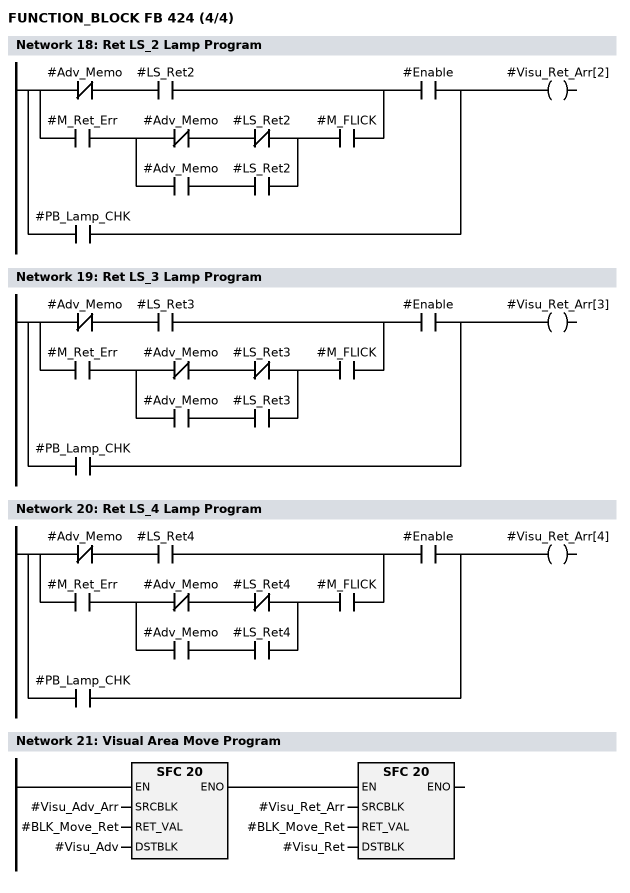
      A(    ;
      AN    #Adv_Memo;
      A     #LS_Ret2;
      O     ;
      A     #M_Ret_Err;
      A(    ;
      AN    #Adv_Memo;
      AN    #LS_Ret2;
      O     ;
      A     #Adv_Memo;
      A     #LS_Ret2;
      )     ;
      A     #M_FLICK;
      )     ;
      A     #Enable;
      O     #PB_Lamp_CHK;
      =     #Visu_Ret_Arr[2];
NETWORK
TITLE =Ret LS_3 Lamp Program
//
//
      A(    ;
      AN    #Adv_Memo;
      A     #LS_Ret3;
      O     ;
      A     #M_Ret_Err;
      A(    ;
      AN    #Adv_Memo;
      AN    #LS_Ret3;
      O     ;
      A     #Adv_Memo;
      A     #LS_Ret3;
      )     ;
      A     #M_FLICK;
      )     ;
      A     #Enable;
      O     #PB_Lamp_CHK;
      =     #Visu_Ret_Arr[3];
NETWORK
TITLE =Ret LS_4 Lamp Program
//
//
      A(    ;
      AN    #Adv_Memo;
      A     #LS_Ret4;
      O     ;
      A     #M_Ret_Err;
      A(    ;
      AN    #Adv_Memo;
      AN    #LS_Ret4;
      O     ;
      A     #Adv_Memo;
      A     #LS_Ret4;
      )     ;
      A     #M_FLICK;
      )     ;
      A     #Enable;
      O     #PB_Lamp_CHK;
      =     #Visu_Ret_Arr[4];
NETWORK
TITLE =Visual Area Move Program

      A(    ;
      CALL SFC   20 (
           SRCBLK                   := #Visu_Adv_Arr,
           RET_VAL                  := #BLK_Move_Ret,
           DSTBLK                   := #Visu_Adv);
      A     BR;
      )     ;
      JNB   _001;
      CALL SFC   20 (
           SRCBLK                   := #Visu_Ret_Arr,
           RET_VAL                  := #BLK_Move_Ret,
           DSTBLK                   := #Visu_Ret);
_001: NOP   0;
END_FUNCTION_BLOCK

FUNCTION_BLOCK FB 426
TITLE =Sensor Error,Lamp Variables Program
AUTHOR : HMC
FAMILY : Common
NAME : Common
VERSION : 1.0


VAR_INPUT
  Enable_Aux : BOOL ;
  Adv_Amount : INT ;
  Ret_Amount : INT ;
  LS_Adv1 : BOOL ;
  LS_Ret1 : BOOL ;
  LS_Adv2 : BOOL ;
  LS_Ret2 : BOOL ;
  LS_Adv3 : BOOL ;
  LS_Ret3 : BOOL ;
  LS_Adv4 : BOOL ;
  LS_Ret4 : BOOL ;
  LS_Adv5 : BOOL ;
  LS_Ret5 : BOOL ;
  LS_Adv6 : BOOL ;
  LS_Ret6 : BOOL ;
  LS_Adv7 : BOOL ;
  LS_Ret7 : BOOL ;
  LS_Adv8 : BOOL ;
  LS_Ret8 : BOOL ;
  SOL_Adv : BOOL ;
  SOL_Ret : BOOL ;
  M_Ready : BOOL ;
  T_CHK1 : TIME ;
  T_CHK2 : TIME ;
  PB_Lamp_CHK : BOOL ;
  PB_Error_Rst : BOOL ;
  M_FLICK : BOOL ;
END_VAR
VAR_OUTPUT
  M_Adv_Err : BOOL ;
  M_Ret_Err : BOOL ;
  LP_Adv : BOOL ;
  LP_Ret : BOOL ;
  Visu_Adv : WORD ;
  Visu_Ret : WORD ;
END_VAR
VAR
  Error_T1 : SFB 4;
  Error_T2 : SFB 4;
  Adv_End_Aux : BOOL ;
  Ret_End_Aux : BOOL ;
  CHK_Aux1 : BOOL ;
  CHK_Aux2 : BOOL ;
  Error_T1_DN : BOOL ;
  Error_T2_DN : BOOL ;
  Adv_Memo : BOOL ;
  Visu_Adv_Arr : ARRAY  [0 .. 15 ] OF BOOL ;
  Visu_Ret_Arr : ARRAY  [0 .. 15 ] OF BOOL ;
  BLK_Move_Ret : INT ;
  Enable : BOOL ;
  Adv_End : BOOL ;
  Ret_End : BOOL ;
END_VAR
BEGIN
NETWORK
TITLE =
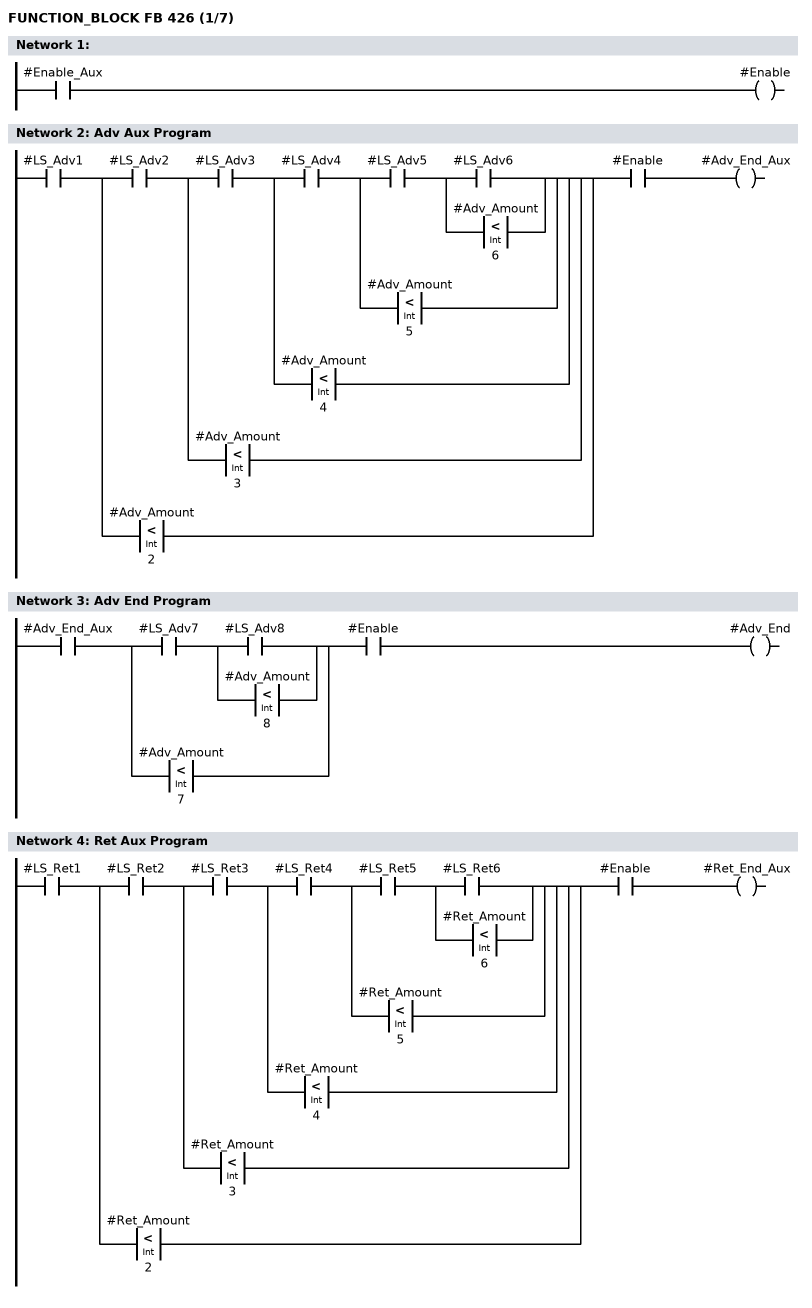

      A     #Enable_Aux;
      =     #Enable;
NETWORK
TITLE =Adv Aux Program

      A     #LS_Adv1;
      A(    ;
      A     #LS_Adv2;
      A(    ;
      A     #LS_Adv3;
      A(    ;
      A     #LS_Adv4;
      A(    ;
      A     #LS_Adv5;
      A(    ;
      O     #LS_Adv6;
      O(    ;
      L     #Adv_Amount;
      L     6;
      <I    ;
      )     ;
      )     ;
      O(    ;
      L     #Adv_Amount;
      L     5;
      <I    ;
      )     ;
      )     ;
      O(    ;
      L     #Adv_Amount;
      L     4;
      <I    ;
      )     ;
      )     ;
      O(    ;
      L     #Adv_Amount;
      L     3;
      <I    ;
      )     ;
      )     ;
      O(    ;
      L     #Adv_Amount;
      L     2;
      <I    ;
      )     ;
      )     ;
      A     #Enable;
      =     #Adv_End_Aux;
NETWORK
TITLE =Adv End Program

      A     #Adv_End_Aux;
      A(    ;
      A     #LS_Adv7;
      A(    ;
      O     #LS_Adv8;
      O(    ;
      L     #Adv_Amount;
      L     8;
      <I    ;
      )     ;
      )     ;
      O(    ;
      L     #Adv_Amount;
      L     7;
      <I    ;
      )     ;
      )     ;
      A     #Enable;
      =     #Adv_End;
NETWORK
TITLE =Ret Aux Program

      A     #LS_Ret1;
      A(    ;
      A     #LS_Ret2;
      A(    ;
      A     #LS_Ret3;
      A(    ;
      A     #LS_Ret4;
      A(    ;
      A     #LS_Ret5;
      A(    ;
      O     #LS_Ret6;
      O(    ;
      L     #Ret_Amount;
      L     6;
      <I    ;
      )     ;
      )     ;
      O(    ;
      L     #Ret_Amount;
      L     5;
      <I    ;
      )     ;
      )     ;
      O(    ;
      L     #Ret_Amount;
      L     4;
      <I    ;
      )     ;
      )     ;
      O(    ;
      L     #Ret_Amount;
      L     3;
      <I    ;
      )     ;
      )     ;
      O(    ;
      L     #Ret_Amount;
      L     2;
      <I    ;
      )     ;
      )     ;
      A     #Enable;
      =     #Ret_End_Aux;
NETWORK
TITLE =Ret End Program
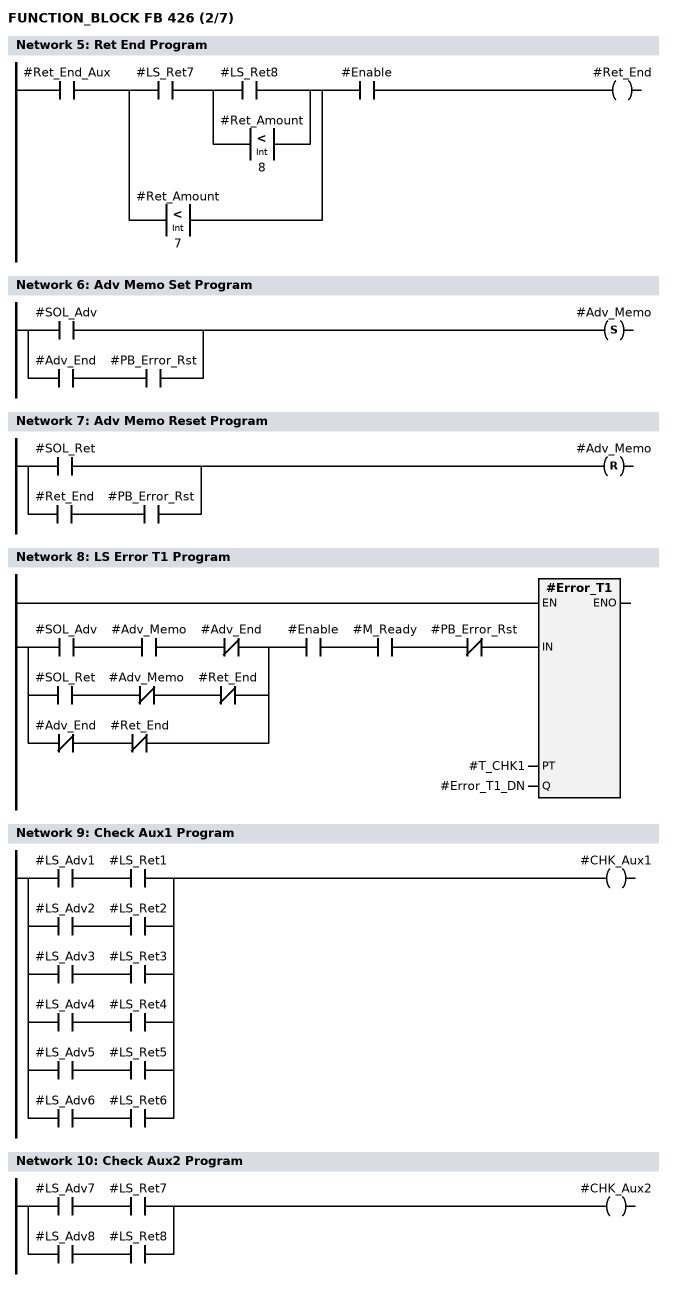

      A     #Ret_End_Aux;
      A(    ;
      A     #LS_Ret7;
      A(    ;
      O     #LS_Ret8;
      O(    ;
      L     #Ret_Amount;
      L     8;
      <I    ;
      )     ;
      )     ;
      O(    ;
      L     #Ret_Amount;
      L     7;
      <I    ;
      )     ;
      )     ;
      A     #Enable;
      =     #Ret_End;
NETWORK
TITLE =Adv Memo Set Program

      O     #SOL_Adv;
      O     ;
      A     #Adv_End;
      A     #PB_Error_Rst;
      S     #Adv_Memo;
NETWORK
TITLE =Adv Memo Reset Program

      O     #SOL_Ret;
      O     ;
      A     #Ret_End;
      A     #PB_Error_Rst;
      R     #Adv_Memo;
NETWORK
TITLE =LS Error T1 Program

      A(    ;
      A     #SOL_Adv;
      A     #Adv_Memo;
      AN    #Adv_End;
      O     ;
      A     #SOL_Ret;
      AN    #Adv_Memo;
      AN    #Ret_End;
      O     ;
      AN    #Adv_End;
      AN    #Ret_End;
      )     ;
      A     #Enable;
      A     #M_Ready;
      AN    #PB_Error_Rst;
      =     L      0.0;
      BLD   103;
      CALL #Error_T1 (
           IN                       := L      0.0,
           PT                       := #T_CHK1,
           Q                        := #Error_T1_DN);

      NOP   0;
NETWORK
TITLE =Check Aux1 Program

      A     #LS_Adv1;
      A     #LS_Ret1;
      O     ;
      A     #LS_Adv2;
      A     #LS_Ret2;
      O     ;
      A     #LS_Adv3;
      A     #LS_Ret3;
      O     ;
      A     #LS_Adv4;
      A     #LS_Ret4;
      O     ;
      A     #LS_Adv5;
      A     #LS_Ret5;
      O     ;
      A     #LS_Adv6;
      A     #LS_Ret6;
      =     #CHK_Aux1;
NETWORK
TITLE =Check Aux2 Program

      A     #LS_Adv7;
      A     #LS_Ret7;
      O     ;
      A     #LS_Adv8;
      A     #LS_Ret8;
      =     #CHK_Aux2;
NETWORK
TITLE =LS Error T2 Program
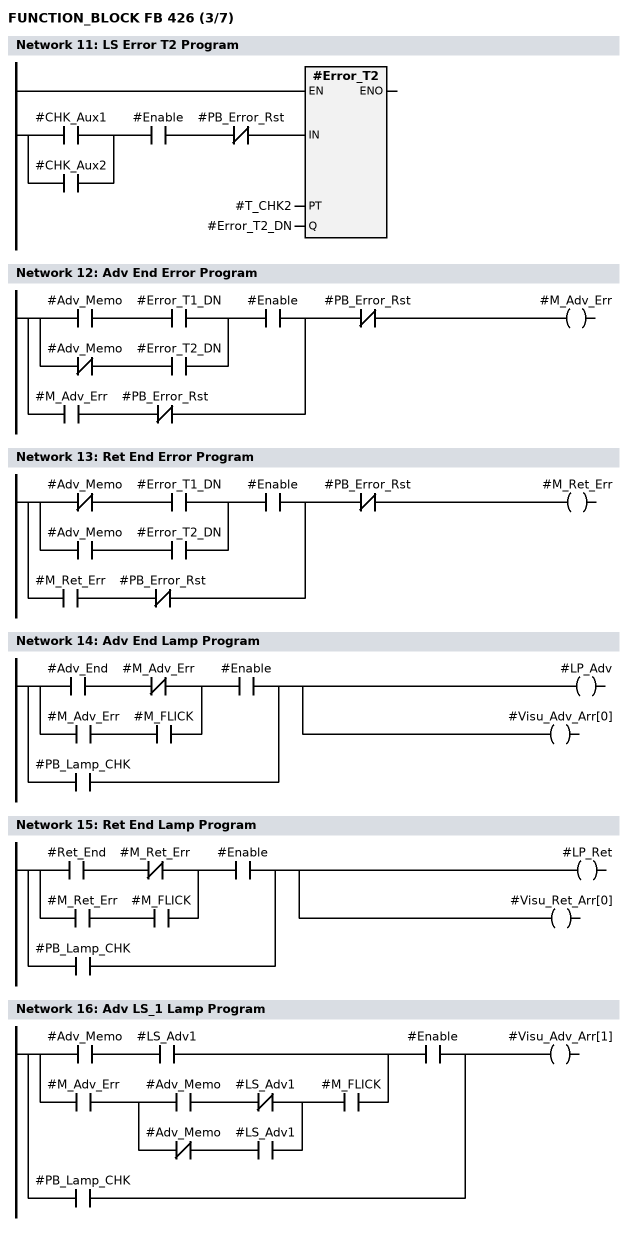

      A(    ;
      O     #CHK_Aux1;
      O     #CHK_Aux2;
      )     ;
      A     #Enable;
      AN    #PB_Error_Rst;
      =     L      0.0;
      BLD   103;
      CALL #Error_T2 (
           IN                       := L      0.0,
           PT                       := #T_CHK2,
           Q                        := #Error_T2_DN);

      NOP   0;
NETWORK
TITLE =Adv End Error Program

      A(    ;
      A(    ;
      A     #Adv_Memo;
      A     #Error_T1_DN;
      O     ;
      AN    #Adv_Memo;
      A     #Error_T2_DN;
      )     ;
      A     #Enable;
      O     ;
      A     #M_Adv_Err;
      AN    #PB_Error_Rst;
      )     ;
      AN    #PB_Error_Rst;
      =     #M_Adv_Err;
NETWORK
TITLE =Ret End Error Program

      A(    ;
      A(    ;
      AN    #Adv_Memo;
      A     #Error_T1_DN;
      O     ;
      A     #Adv_Memo;
      A     #Error_T2_DN;
      )     ;
      A     #Enable;
      O     ;
      A     #M_Ret_Err;
      AN    #PB_Error_Rst;
      )     ;
      AN    #PB_Error_Rst;
      =     #M_Ret_Err;
NETWORK
TITLE =Adv End Lamp Program

      A(    ;
      A     #Adv_End;
      AN    #M_Adv_Err;
      O     ;
      A     #M_Adv_Err;
      A     #M_FLICK;
      )     ;
      A     #Enable;
      O     #PB_Lamp_CHK;
      =     #LP_Adv;
      =     #Visu_Adv_Arr[0];
NETWORK
TITLE =Ret End Lamp Program

      A(    ;
      A     #Ret_End;
      AN    #M_Ret_Err;
      O     ;
      A     #M_Ret_Err;
      A     #M_FLICK;
      )     ;
      A     #Enable;
      O     #PB_Lamp_CHK;
      =     #LP_Ret;
      =     #Visu_Ret_Arr[0];
NETWORK
TITLE =Adv LS_1 Lamp Program

      A(    ;
      A     #Adv_Memo;
      A     #LS_Adv1;
      O     ;
      A     #M_Adv_Err;
      A(    ;
      A     #Adv_Memo;
      AN    #LS_Adv1;
      O     ;
      AN    #Adv_Memo;
      A     #LS_Adv1;
      )     ;
      A     #M_FLICK;
      )     ;
      A     #Enable;
      O     #PB_Lamp_CHK;
      =     #Visu_Adv_Arr[1];
NETWORK
TITLE =Adv LS_2 Lamp Program
//
//
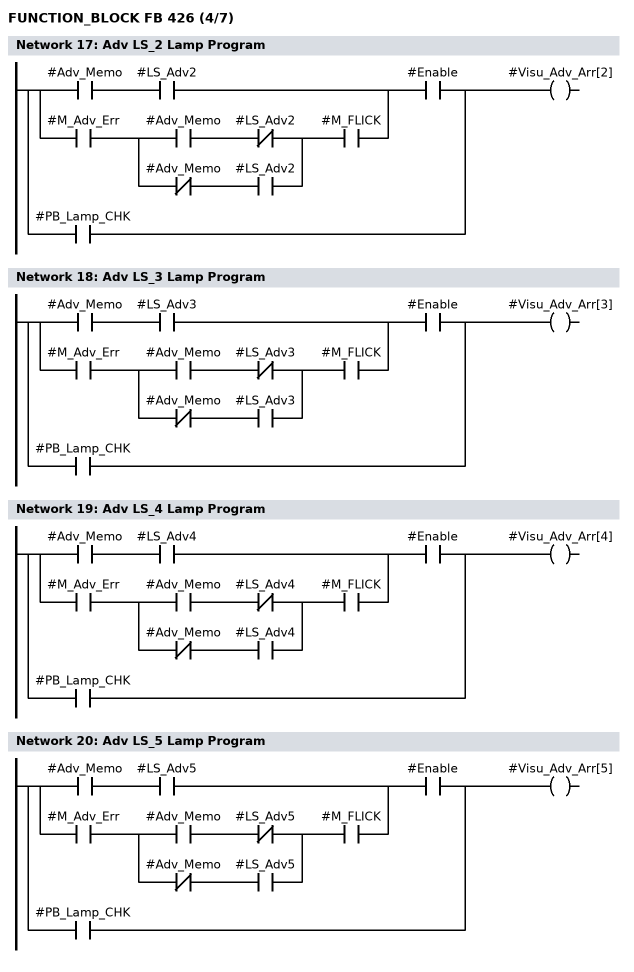
      A(    ;
      A     #Adv_Memo;
      A     #LS_Adv2;
      O     ;
      A     #M_Adv_Err;
      A(    ;
      A     #Adv_Memo;
      AN    #LS_Adv2;
      O     ;
      AN    #Adv_Memo;
      A     #LS_Adv2;
      )     ;
      A     #M_FLICK;
      )     ;
      A     #Enable;
      O     #PB_Lamp_CHK;
      =     #Visu_Adv_Arr[2];
NETWORK
TITLE =Adv LS_3 Lamp Program
//
//
      A(    ;
      A     #Adv_Memo;
      A     #LS_Adv3;
      O     ;
      A     #M_Adv_Err;
      A(    ;
      A     #Adv_Memo;
      AN    #LS_Adv3;
      O     ;
      AN    #Adv_Memo;
      A     #LS_Adv3;
      )     ;
      A     #M_FLICK;
      )     ;
      A     #Enable;
      O     #PB_Lamp_CHK;
      =     #Visu_Adv_Arr[3];
NETWORK
TITLE =Adv LS_4 Lamp Program
//
//
      A(    ;
      A     #Adv_Memo;
      A     #LS_Adv4;
      O     ;
      A     #M_Adv_Err;
      A(    ;
      A     #Adv_Memo;
      AN    #LS_Adv4;
      O     ;
      AN    #Adv_Memo;
      A     #LS_Adv4;
      )     ;
      A     #M_FLICK;
      )     ;
      A     #Enable;
      O     #PB_Lamp_CHK;
      =     #Visu_Adv_Arr[4];
NETWORK
TITLE =Adv LS_5 Lamp Program
//
//
      A(    ;
      A     #Adv_Memo;
      A     #LS_Adv5;
      O     ;
      A     #M_Adv_Err;
      A(    ;
      A     #Adv_Memo;
      AN    #LS_Adv5;
      O     ;
      AN    #Adv_Memo;
      A     #LS_Adv5;
      )     ;
      A     #M_FLICK;
      )     ;
      A     #Enable;
      O     #PB_Lamp_CHK;
      =     #Visu_Adv_Arr[5];
NETWORK
TITLE =Adv LS_6 Lamp Program
//
//
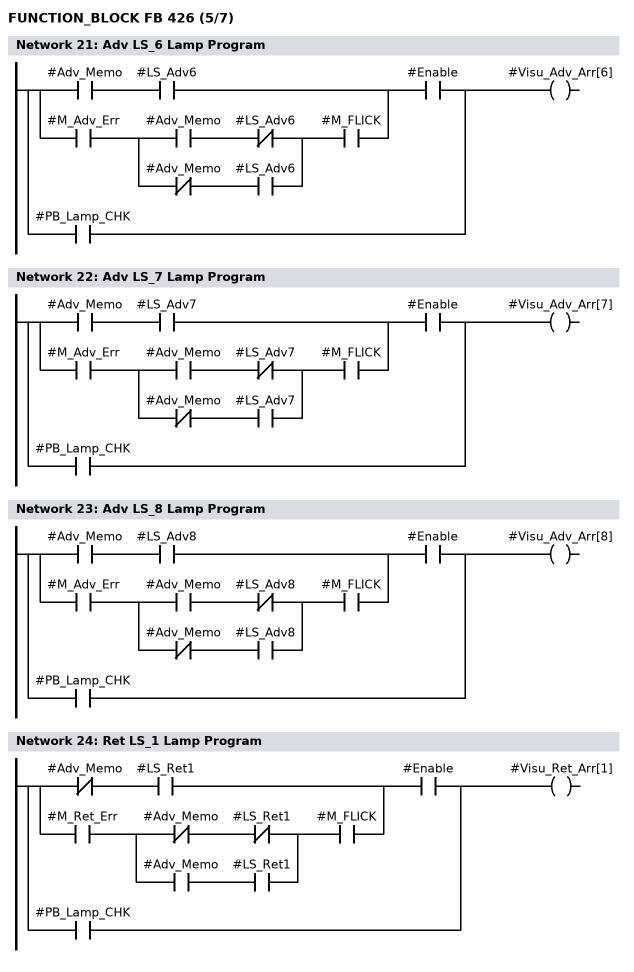
      A(    ;
      A     #Adv_Memo;
      A     #LS_Adv6;
      O     ;
      A     #M_Adv_Err;
      A(    ;
      A     #Adv_Memo;
      AN    #LS_Adv6;
      O     ;
      AN    #Adv_Memo;
      A     #LS_Adv6;
      )     ;
      A     #M_FLICK;
      )     ;
      A     #Enable;
      O     #PB_Lamp_CHK;
      =     #Visu_Adv_Arr[6];
NETWORK
TITLE =Adv LS_7 Lamp Program
//
//
      A(    ;
      A     #Adv_Memo;
      A     #LS_Adv7;
      O     ;
      A     #M_Adv_Err;
      A(    ;
      A     #Adv_Memo;
      AN    #LS_Adv7;
      O     ;
      AN    #Adv_Memo;
      A     #LS_Adv7;
      )     ;
      A     #M_FLICK;
      )     ;
      A     #Enable;
      O     #PB_Lamp_CHK;
      =     #Visu_Adv_Arr[7];
NETWORK
TITLE =Adv LS_8 Lamp Program
//
//
      A(    ;
      A     #Adv_Memo;
      A     #LS_Adv8;
      O     ;
      A     #M_Adv_Err;
      A(    ;
      A     #Adv_Memo;
      AN    #LS_Adv8;
      O     ;
      AN    #Adv_Memo;
      A     #LS_Adv8;
      )     ;
      A     #M_FLICK;
      )     ;
      A     #Enable;
      O     #PB_Lamp_CHK;
      =     #Visu_Adv_Arr[8];
NETWORK
TITLE =Ret LS_1 Lamp Program
//
//
      A(    ;
      AN    #Adv_Memo;
      A     #LS_Ret1;
      O     ;
      A     #M_Ret_Err;
      A(    ;
      AN    #Adv_Memo;
      AN    #LS_Ret1;
      O     ;
      A     #Adv_Memo;
      A     #LS_Ret1;
      )     ;
      A     #M_FLICK;
      )     ;
      A     #Enable;
      O     #PB_Lamp_CHK;
      =     #Visu_Ret_Arr[1];
NETWORK
TITLE =Ret LS_2 Lamp Program
//
//
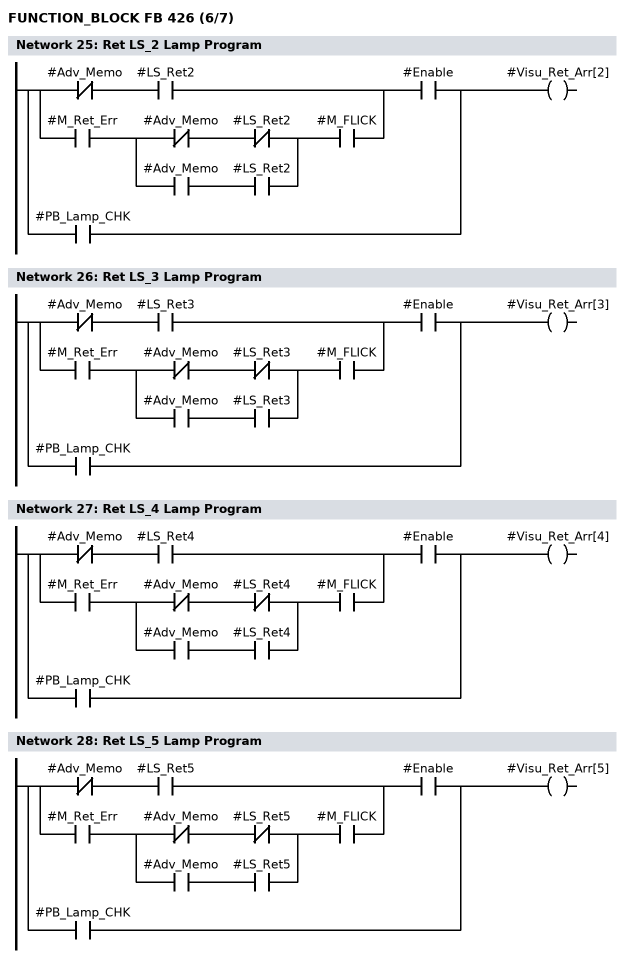
      A(    ;
      AN    #Adv_Memo;
      A     #LS_Ret2;
      O     ;
      A     #M_Ret_Err;
      A(    ;
      AN    #Adv_Memo;
      AN    #LS_Ret2;
      O     ;
      A     #Adv_Memo;
      A     #LS_Ret2;
      )     ;
      A     #M_FLICK;
      )     ;
      A     #Enable;
      O     #PB_Lamp_CHK;
      =     #Visu_Ret_Arr[2];
NETWORK
TITLE =Ret LS_3 Lamp Program
//
//
      A(    ;
      AN    #Adv_Memo;
      A     #LS_Ret3;
      O     ;
      A     #M_Ret_Err;
      A(    ;
      AN    #Adv_Memo;
      AN    #LS_Ret3;
      O     ;
      A     #Adv_Memo;
      A     #LS_Ret3;
      )     ;
      A     #M_FLICK;
      )     ;
      A     #Enable;
      O     #PB_Lamp_CHK;
      =     #Visu_Ret_Arr[3];
NETWORK
TITLE =Ret LS_4 Lamp Program
//
//
      A(    ;
      AN    #Adv_Memo;
      A     #LS_Ret4;
      O     ;
      A     #M_Ret_Err;
      A(    ;
      AN    #Adv_Memo;
      AN    #LS_Ret4;
      O     ;
      A     #Adv_Memo;
      A     #LS_Ret4;
      )     ;
      A     #M_FLICK;
      )     ;
      A     #Enable;
      O     #PB_Lamp_CHK;
      =     #Visu_Ret_Arr[4];
NETWORK
TITLE =Ret LS_5 Lamp Program
//
//
      A(    ;
      AN    #Adv_Memo;
      A     #LS_Ret5;
      O     ;
      A     #M_Ret_Err;
      A(    ;
      AN    #Adv_Memo;
      AN    #LS_Ret5;
      O     ;
      A     #Adv_Memo;
      A     #LS_Ret5;
      )     ;
      A     #M_FLICK;
      )     ;
      A     #Enable;
      O     #PB_Lamp_CHK;
      =     #Visu_Ret_Arr[5];
NETWORK
TITLE =Ret LS_6 Lamp Program
//
//
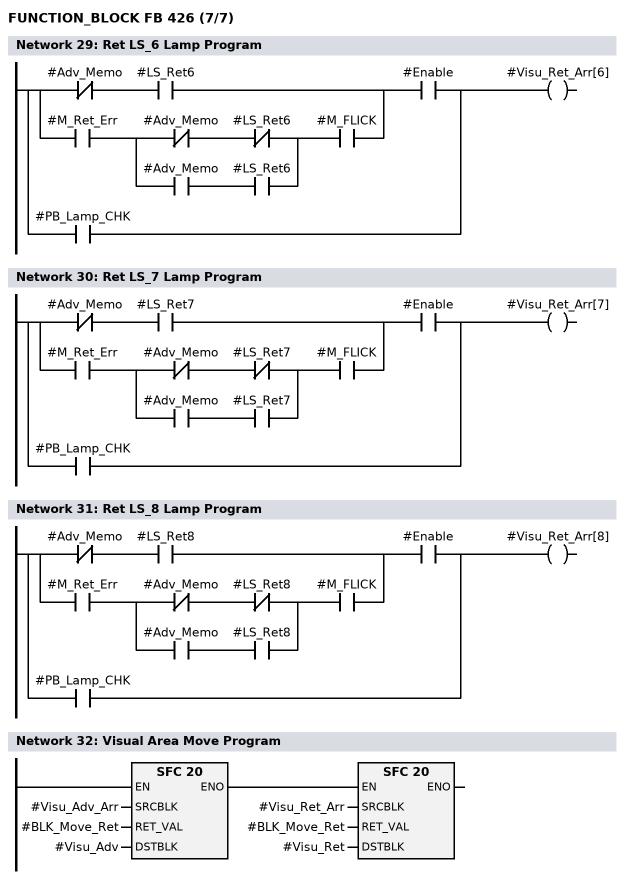
      A(    ;
      AN    #Adv_Memo;
      A     #LS_Ret6;
      O     ;
      A     #M_Ret_Err;
      A(    ;
      AN    #Adv_Memo;
      AN    #LS_Ret6;
      O     ;
      A     #Adv_Memo;
      A     #LS_Ret6;
      )     ;
      A     #M_FLICK;
      )     ;
      A     #Enable;
      O     #PB_Lamp_CHK;
      =     #Visu_Ret_Arr[6];
NETWORK
TITLE =Ret LS_7 Lamp Program
//
//
      A(    ;
      AN    #Adv_Memo;
      A     #LS_Ret7;
      O     ;
      A     #M_Ret_Err;
      A(    ;
      AN    #Adv_Memo;
      AN    #LS_Ret7;
      O     ;
      A     #Adv_Memo;
      A     #LS_Ret7;
      )     ;
      A     #M_FLICK;
      )     ;
      A     #Enable;
      O     #PB_Lamp_CHK;
      =     #Visu_Ret_Arr[7];
NETWORK
TITLE =Ret LS_8 Lamp Program
//
//
      A(    ;
      AN    #Adv_Memo;
      A     #LS_Ret8;
      O     ;
      A     #M_Ret_Err;
      A(    ;
      AN    #Adv_Memo;
      AN    #LS_Ret8;
      O     ;
      A     #Adv_Memo;
      A     #LS_Ret8;
      )     ;
      A     #M_FLICK;
      )     ;
      A     #Enable;
      O     #PB_Lamp_CHK;
      =     #Visu_Ret_Arr[8];
NETWORK
TITLE =Visual Area Move Program

      A(    ;
      CALL SFC   20 (
           SRCBLK                   := #Visu_Adv_Arr,
           RET_VAL                  := #BLK_Move_Ret,
           DSTBLK                   := #Visu_Adv);
      A     BR;
      )     ;
      JNB   _001;
      CALL SFC   20 (
           SRCBLK                   := #Visu_Ret_Arr,
           RET_VAL                  := #BLK_Move_Ret,
           DSTBLK                   := #Visu_Ret);
_001: NOP   0;
END_FUNCTION_BLOCK

FUNCTION_BLOCK FB 500
TITLE =CYCLE TIME CHECK
VERSION : 0.1


VAR_INPUT
  CYCLE_UP : BOOL ;
  CYCLE_RST : BOOL ;
END_VAR
VAR_OUTPUT
  CURRENT_CT : INT ;
  PREVIOUS_CT : INT ;
END_VAR
VAR
  CURRENT : INT ;
  PREVIOUS : INT ;
  CYCLE_UP_PLS : BOOL ;
  CYCLE_RST_PLS : BOOL ;
  CYCLE_OVER_PLS : BOOL ;
END_VAR
BEGIN
NETWORK
TITLE =CURRENT TIME CHK
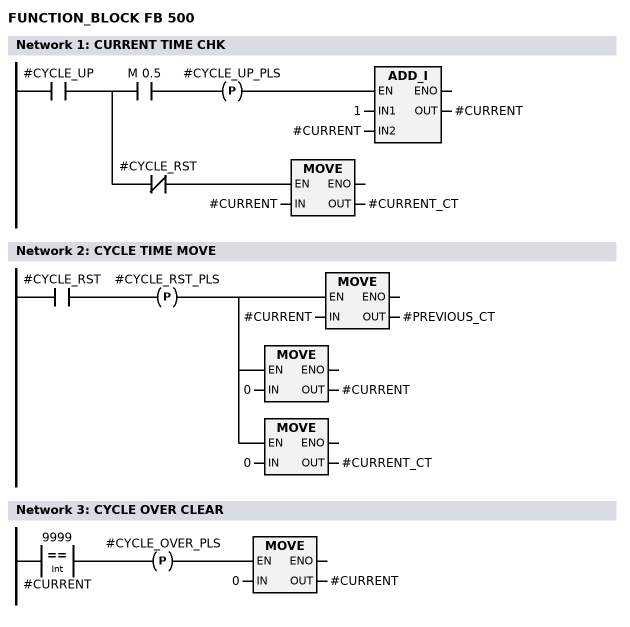

      A     #CYCLE_UP;
      =     L      0.0;
      A     L      0.0;
      A     M      0.5;
      FP    #CYCLE_UP_PLS;
      JNB   _001;
      L     1;
      L     #CURRENT;
      +I    ;
      T     #CURRENT;
_001: NOP   0;
      A     L      0.0;
      AN    #CYCLE_RST;
      JNB   _002;
      L     #CURRENT;
      T     #CURRENT_CT;
_002: NOP   0;
NETWORK
TITLE =CYCLE TIME MOVE

      A     #CYCLE_RST;
      FP    #CYCLE_RST_PLS;
      =     L      0.0;
      A     L      0.0;
      JNB   _003;
      L     #CURRENT;
      T     #PREVIOUS_CT;
_003: NOP   0;
      A     L      0.0;
      JNB   _004;
      L     0;
      T     #CURRENT;
_004: NOP   0;
      A     L      0.0;
      JNB   _005;
      L     0;
      T     #CURRENT_CT;
_005: NOP   0;
NETWORK
TITLE =CYCLE OVER CLEAR

      A(    ;
      L     9999;
      L     #CURRENT;
      ==I   ;
      )     ;
      FP    #CYCLE_OVER_PLS;
      JNB   _006;
      L     0;
      T     #CURRENT;
_006: NOP   0;
END_FUNCTION_BLOCK

FUNCTION FC 98 : VOID
TITLE =
VERSION : 0.1


VAR_TEMP
  SFC20_RET_VAL : INT ;
  RECV1_LEN : WORD ;
  SEND1_LEN : WORD ;
  RECV2_LEN : WORD ;
  SEND2_LEN : WORD ;
END_VAR
BEGIN
NETWORK
TITLE =
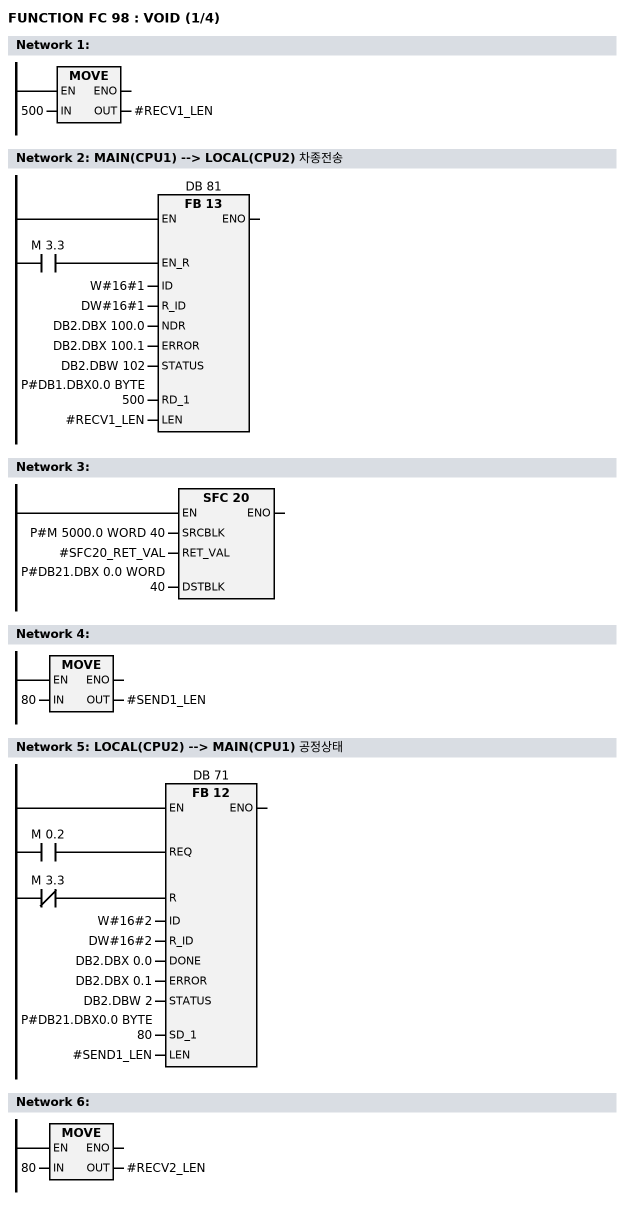

      L     500;
      T     #RECV1_LEN;
      NOP   0;
NETWORK
TITLE =MAIN(CPU1) --> LOCAL(CPU2) 차종전송

